# B&R Automation Studio project RobotNewEra (part 8)

### Data object Logical/MotionHandling/MotionInitFiles/SDC/sdc_j5_i (Ax)

#### sdc_j5_i.ax
```
InitParameter (Version=2.46.0, NcSwId=ACP10)
  ACP10AXIS_typ:
    dig_in:
      level:
        reference = ncACTIV_HI
        pos_hw_end = ncACTIV_HI
        neg_hw_end = ncACTIV_HI
        trigger1 = ncACTIV_HI
        trigger2 = ncACTIV_LO + ncQUICKSTOP
    encoder_if:
      parameter:
        count_dir = ncSTANDARD
        scaling:
          load:
            units = 360000
            rev_motor = 119
    limit:
      parameter:
        v_pos = 120000.0
        v_neg = 120000.0
        a1_pos = 240000.0
        a2_pos = 240000.0
        a1_neg = 240000.0
        a2_neg = 240000.0
        t_jolt = 0.1
        t_in_pos = 0.0
        pos_sw_end = 125000
        neg_sw_end = -125000
        ds_warning = 5000.0
        ds_stop = 10000.0
        a_stop = 1.0e+30
        dv_stop = 0.0
        dv_stop_mode = ncOFF
    controller:
      mode = ncPOSITION
      position:
        kv = 560.0
        tn = 0.0
        t_predict = 0.0004
        t_total = 0.0004
        p_max = 1.0e+30
        i_max = 20000.0
      speed:
        kv = 29.3
        tn = 0.0
        t_filter = 0.0
        isq_filter1:
          type = ncOFF
          a0 = 0.0
          a1 = 0.0
          b0 = 0.0
          b1 = 0.0
          b2 = 0.0
          c0_par_id = 0
          c1_par_id = 0
        isq_filter2:
          type = ncOFF
          a0 = 0.0
          a1 = 0.0
          b0 = 0.0
          b1 = 0.0
          b2 = 0.0
          c0_par_id = 0
          c1_par_id = 0
        isq_filter3:
          type = ncOFF
          a0 = 0.0
          a1 = 0.0
          b0 = 0.0
          b1 = 0.0
          b2 = 0.0
          c0_par_id = 0
          c1_par_id = 0
      uf:
        type = ncLINEAR
        auto_config = ncMOTOR_PAR
        u0 = 0.0
        un = 0.0
        fn = 50.0
        k_f_slip = 0.0
      ff:
        torque_load = 0.0
        torque_pos = 0.0
        torque_neg = 0.0
        kv_torque = 0.0
        inertia = 0.0
        t_filter_a = 0.0
    move:
      stop:
        parameter[0]:
          decel_ramp = ncA_LIMIT
          controller = ncON
        parameter[1]:
          decel_ramp = ncA_LIMIT
          controller = ncON
        parameter[2]:
          decel_ramp = ncA_LIMIT
          controller = ncON
        parameter[3]:
          decel_ramp = ncA_LIMIT
          controller = ncON
        quickstop:
          decel_ramp = ncA_LIMIT
        drive_error:
          decel_ramp = ncA_LIMIT
      homing:
        parameter:
          s = 0
          v_switch = 5000.0
          v_trigger = 500.0
          a = 50000.0
          mode = ncDIRECT
          edge_sw = ncPOSITIVE
          start_dir = ncPOSITIVE
          trigg_dir = ncPOSITIVE
          ref_pulse = ncOFF
          fix_dir = ncOFF
          tr_s_block = 0.0
          torque_lim = 0.0
          ds_block = 0.0
          ds_stop = 0.0
      basis:
        parameter:
          v_pos = 5000.0
          v_neg = 5000.0
          a1_pos = 100000.0
          a2_pos = 100000.0
          a1_neg = 100000.0
          a2_neg = 100000.0
    message:
      text:
        parameter:
          format = ncBREAK
          columns = 80
          data_modul = AcpError
```

### Data object Logical/MotionHandling/MotionInitFiles/SDC/sdc_j6_i (Ax)

#### sdc_j6_i.ax
```
InitParameter (Version=2.46.0, NcSwId=ACP10)
  ACP10AXIS_typ:
    dig_in:
      level:
        reference = ncACTIV_HI
        pos_hw_end = ncACTIV_HI
        neg_hw_end = ncACTIV_HI
        trigger1 = ncACTIV_HI
        trigger2 = ncACTIV_LO + ncQUICKSTOP
    encoder_if:
      parameter:
        count_dir = ncSTANDARD
        scaling:
          load:
            units = 360000
            rev_motor = 89
    limit:
      parameter:
        v_pos = 190000.0
        v_neg = 190000.0
        a1_pos = 380000.0
        a2_pos = 380000.0
        a1_neg = 380000.0
        a2_neg = 380000.0
        t_jolt = 0.1
        t_in_pos = 0.0
        pos_sw_end = 360000
        neg_sw_end = -360000
        ds_warning = 5000.0
        ds_stop = 10000.0
        a_stop = 1.0e+30
        dv_stop = 0.0
        dv_stop_mode = ncOFF
    controller:
      mode = ncPOSITION
      position:
        kv = 540.0
        tn = 0.0
        t_predict = 0.0004
        t_total = 0.0004
        p_max = 1.0e+30
        i_max = 2000.0
      speed:
        kv = 29.85
        tn = 0.0
        t_filter = 0.0
        isq_filter1:
          type = ncOFF
          a0 = 0.0
          a1 = 0.0
          b0 = 0.0
          b1 = 0.0
          b2 = 0.0
          c0_par_id = 0
          c1_par_id = 0
        isq_filter2:
          type = ncOFF
          a0 = 0.0
          a1 = 0.0
          b0 = 0.0
          b1 = 0.0
          b2 = 0.0
          c0_par_id = 0
          c1_par_id = 0
        isq_filter3:
          type = ncOFF
          a0 = 0.0
          a1 = 0.0
          b0 = 0.0
          b1 = 0.0
          b2 = 0.0
          c0_par_id = 0
          c1_par_id = 0
      uf:
        type = ncLINEAR
        auto_config = ncMOTOR_PAR
        u0 = 0.0
        un = 0.0
        fn = 50.0
        k_f_slip = 0.0
      ff:
        torque_load = 0.00094268
        torque_pos = 0.110223
        torque_neg = 0.100704
        kv_torque = 0.00253262
        inertia = 5.79039e-05
        t_filter_a = 0.0
    move:
      stop:
        parameter[0]:
          decel_ramp = ncA_LIMIT
          controller = ncON
        parameter[1]:
          decel_ramp = ncA_LIMIT
          controller = ncON
        parameter[2]:
          decel_ramp = ncA_LIMIT
          controller = ncON
        parameter[3]:
          decel_ramp = ncA_LIMIT
          controller = ncON
        quickstop:
          decel_ramp = ncA_LIMIT
        drive_error:
          decel_ramp = ncA_LIMIT
      homing:
        parameter:
          s = 0
          v_switch = 5000.0
          v_trigger = 500.0
          a = 50000.0
          mode = ncDIRECT
          edge_sw = ncPOSITIVE
          start_dir = ncPOSITIVE
          trigg_dir = ncPOSITIVE
          ref_pulse = ncOFF
          fix_dir = ncOFF
          tr_s_block = 0.0
          torque_lim = 0.0
          ds_block = 0.0
          ds_stop = 0.0
      basis:
        parameter:
          v_pos = 5000.0
          v_neg = 5000.0
          a1_pos = 100000.0
          a2_pos = 100000.0
          a1_neg = 100000.0
          a2_neg = 100000.0
    message:
      text:
        parameter:
          format = ncBREAK
          columns = 80
          data_modul = AcpError
```

### Data object Logical/MotionHandling/MotionInitFiles/robot_i (Cns) - ARNC0: CNC-System

- robot_i.cns (not shown)

### Package Logical/MotionHandling/Transformations - Trf Related

### Program Logical/MotionHandling/Transformations/Trf (ANSIC)

#### Trf.c - Implementation code
```c
/********************************************************************
 * COPYRIGHT -- Bernecker + Rainer
 ********************************************************************
 * Program: Trf
 * File: Trf.c
 * Author: frigenif
 * Created: December 08, 2011
 ********************************************************************
 * Implementation of program Trf
 ********************************************************************/

#include <bur/plctypes.h>
#include <TRF_LIB.h>

#ifdef _DEFAULT_INCLUDES
 #include <AsDefault.h>
#endif

void _INIT TrfINIT( void )
{

	/* Trasformation Configuration */

	/* Unit definintion */
	Robot_TRF.units.measure= TRF_DEGREES;
	Robot_TRF.units.epsilon= 0.000001;
	// Initialization
	// Warning: Delete those if = 0 then = ,they are only for Testpurpose
	if (HmiRetain.HmiRobot.CartesianLimits[0].Min == 0) HmiRetain.HmiRobot.CartesianLimits[0].Min = -2658;
	if (HmiRetain.HmiRobot.CartesianLimits[1].Min == 0) HmiRetain.HmiRobot.CartesianLimits[1].Min = -2658;
	if (HmiRetain.HmiRobot.CartesianLimits[2].Min == 0) HmiRetain.HmiRobot.CartesianLimits[2].Min = -602;
	if (HmiRetain.HmiRobot.CartesianLimits[0].Max == 0) HmiRetain.HmiRobot.CartesianLimits[0].Max = 2658;
	if (HmiRetain.HmiRobot.CartesianLimits[1].Max == 0) HmiRetain.HmiRobot.CartesianLimits[1].Max = 2658;
	if (HmiRetain.HmiRobot.CartesianLimits[2].Max == 0) HmiRetain.HmiRobot.CartesianLimits[2].Max = 3297;

	if (HmiRetain.HmiRobot.HomePos.Pos.x == 0) HmiRetain.HmiRobot.HomePos.Pos.x = 1854;
	if (HmiRetain.HmiRobot.HomePos.Pos.y == 0) HmiRetain.HmiRobot.HomePos.Pos.y = 0;
	if (HmiRetain.HmiRobot.HomePos.Pos.z == 0) HmiRetain.HmiRobot.HomePos.Pos.z = 1990;

	//	 Dimensions and position in the global coordinate system
	if (HmiRetain.HmiRobot.Mech[1].OffsetX == 0) HmiRetain.HmiRobot.Mech[1].OffsetX = 312.0;
	if (HmiRetain.HmiRobot.Mech[1].OffsetZ == 0) HmiRetain.HmiRobot.Mech[1].OffsetZ = 680.0;
	if (HmiRetain.HmiRobot.Mech[2].OffsetZ == 0) HmiRetain.HmiRobot.Mech[2].OffsetZ = 1075.0;
	if (HmiRetain.HmiRobot.Mech[3].OffsetX == 0) HmiRetain.HmiRobot.Mech[3].OffsetX = 400.0;
	if (HmiRetain.HmiRobot.Mech[3].OffsetZ == 0) HmiRetain.HmiRobot.Mech[3].OffsetZ = 235.0;
	if (HmiRetain.HmiRobot.Mech[4].OffsetX == 0) HmiRetain.HmiRobot.Mech[4].OffsetX = 882.0;
	if (HmiRetain.HmiRobot.Mech[5].OffsetX == 0) HmiRetain.HmiRobot.Mech[5].OffsetX = 260.0;

	Robot_TRF.mech.a0x = HmiRetain.HmiRobot.Mech[0].OffsetX;
	Robot_TRF.mech.a0y = HmiRetain.HmiRobot.Mech[0].OffsetY;
	Robot_TRF.mech.a0z = HmiRetain.HmiRobot.Mech[0].OffsetZ;
	Robot_TRF.mech.a1x = HmiRetain.HmiRobot.Mech[1].OffsetX;
	Robot_TRF.mech.a1y = HmiRetain.HmiRobot.Mech[1].OffsetY;
	Robot_TRF.mech.a1z = HmiRetain.HmiRobot.Mech[1].OffsetZ;
	Robot_TRF.mech.a2x = HmiRetain.HmiRobot.Mech[2].OffsetX;
	Robot_TRF.mech.a2y = HmiRetain.HmiRobot.Mech[2].OffsetY;
	Robot_TRF.mech.a2z = HmiRetain.HmiRobot.Mech[2].OffsetZ;
	Robot_TRF.mech.a3x = HmiRetain.HmiRobot.Mech[3].OffsetX;
	Robot_TRF.mech.a3y = HmiRetain.HmiRobot.Mech[3].OffsetY;
	Robot_TRF.mech.a3z = HmiRetain.HmiRobot.Mech[3].OffsetZ;
	Robot_TRF.mech.a4x = HmiRetain.HmiRobot.Mech[4].OffsetX;
	Robot_TRF.mech.a5x = HmiRetain.HmiRobot.Mech[5].OffsetX;

	Robot_TRF.mech.angles_type = TRF_CARDAN_ANGLES;

	/* preferred mode */
	Robot_TRF.mode.preferred = TRF_MODE_FRONT + TRF_MODE_CONVEX + TRF_MODE_POSITIVE;

	// Joint properties
	if (HmiRetain.HmiRobot.Mech[1].Direction == 0) HmiRetain.HmiRobot.Mech[1].Direction = 1;
	if (HmiRetain.HmiRobot.Mech[2].Direction == 0) HmiRetain.HmiRobot.Mech[2].Direction = 1;
	if (HmiRetain.HmiRobot.Mech[4].Direction == 0) HmiRetain.HmiRobot.Mech[4].Direction = 1;

	if (HmiRetain.HmiRobot.JointLimits[0].Min == 0) HmiRetain.HmiRobot.JointLimits[0].Min = -180;
	if (HmiRetain.HmiRobot.JointLimits[0].Max == 0) HmiRetain.HmiRobot.JointLimits[0].Max = 180;
	if (HmiRetain.HmiRobot.JointLimits[1].Min == 0) HmiRetain.HmiRobot.JointLimits[1].Min = -76;
	if (HmiRetain.HmiRobot.JointLimits[1].Max == 0) HmiRetain.HmiRobot.JointLimits[1].Max = 60;
	if (HmiRetain.HmiRobot.JointLimits[2].Min == 0) HmiRetain.HmiRobot.JointLimits[2].Min = -65; //-142;
	if (HmiRetain.HmiRobot.JointLimits[2].Max == 0) HmiRetain.HmiRobot.JointLimits[2].Max = 230;
	if (HmiRetain.HmiRobot.JointLimits[3].Min == 0) HmiRetain.HmiRobot.JointLimits[3].Min = -360;
	if (HmiRetain.HmiRobot.JointLimits[3].Max == 0) HmiRetain.HmiRobot.JointLimits[3].Max = 360; //-360;
	if (HmiRetain.HmiRobot.JointLimits[4].Min == 0) HmiRetain.HmiRobot.JointLimits[4].Min = -125;
	if (HmiRetain.HmiRobot.JointLimits[4].Max == 0) HmiRetain.HmiRobot.JointLimits[4].Max = 125;
	if (HmiRetain.HmiRobot.JointLimits[5].Min == 0) HmiRetain.HmiRobot.JointLimits[5].Min = -360;
	if (HmiRetain.HmiRobot.JointLimits[5].Max == 0) HmiRetain.HmiRobot.JointLimits[5].Max = 360;

	Robot_TRF.mech.axis_Q1.property = TRF_MATH_POSITIVE + HmiRetain.HmiRobot.Mech[0].Direction + TRF_SW_ENDS_ENABLE + TRF_MULT_FACTOR_DISABLE;
	Robot_TRF.mech.axis_Q1.min_sw_end = HmiRetain.HmiRobot.JointLimits[0].Min;
	Robot_TRF.mech.axis_Q1.max_sw_end = HmiRetain.HmiRobot.JointLimits[0].Max;
	Robot_TRF.mech.axis_Q1.maximal_change = 5000.0;	// obsolete
	Robot_TRF.mech.axis_Q1.mult_factor = 0.0;

	Robot_TRF.mech.axis_Q2.property = TRF_MATH_POSITIVE + HmiRetain.HmiRobot.Mech[1].Direction + TRF_SW_ENDS_ENABLE + TRF_MULT_FACTOR_DISABLE ;
	Robot_TRF.mech.axis_Q2.min_sw_end = HmiRetain.HmiRobot.JointLimits[1].Min;
	Robot_TRF.mech.axis_Q2.max_sw_end = HmiRetain.HmiRobot.JointLimits[1].Max;
	Robot_TRF.mech.axis_Q2.maximal_change = 5000.0;	// obsolete
	Robot_TRF.mech.axis_Q2.mult_factor = 0.0;

	Robot_TRF.mech.axis_Q3.property = TRF_MATH_POSITIVE + HmiRetain.HmiRobot.Mech[2].Direction + TRF_SW_ENDS_ENABLE + TRF_MULT_FACTOR_DISABLE;
	Robot_TRF.mech.axis_Q3.min_sw_end = HmiRetain.HmiRobot.JointLimits[2].Min;
	Robot_TRF.mech.axis_Q3.max_sw_end = HmiRetain.HmiRobot.JointLimits[2].Max;
	Robot_TRF.mech.axis_Q3.maximal_change = 5000.0;	// obsolete
	Robot_TRF.mech.axis_Q3.mult_factor = 0.0;

	Robot_TRF.mech.axis_Q4.property = TRF_MATH_POSITIVE + HmiRetain.HmiRobot.Mech[3].Direction + TRF_SW_ENDS_ENABLE + TRF_MULT_FACTOR_DISABLE;
	Robot_TRF.mech.axis_Q4.min_sw_end = HmiRetain.HmiRobot.JointLimits[3].Min;
	Robot_TRF.mech.axis_Q4.max_sw_end = HmiRetain.HmiRobot.JointLimits[3].Max;
	Robot_TRF.mech.axis_Q4.maximal_change = 5000.0;	// obsolete
	Robot_TRF.mech.axis_Q4.mult_factor = 0.0;

	Robot_TRF.mech.axis_Q5.property = TRF_MATH_POSITIVE + HmiRetain.HmiRobot.Mech[4].Direction + TRF_SW_ENDS_ENABLE + TRF_MULT_FACTOR_DISABLE;
	Robot_TRF.mech.axis_Q5.min_sw_end = HmiRetain.HmiRobot.JointLimits[4].Min;
	Robot_TRF.mech.axis_Q5.max_sw_end = HmiRetain.HmiRobot.JointLimits[4].Max;
	Robot_TRF.mech.axis_Q5.maximal_change = 5000.0;	// obsolete
	Robot_TRF.mech.axis_Q5.mult_factor = 0.0;

	Robot_TRF.mech.axis_Q6.property = TRF_MATH_POSITIVE + HmiRetain.HmiRobot.Mech[5].Direction + TRF_SW_ENDS_ENABLE + TRF_MULT_FACTOR_DISABLE;
	Robot_TRF.mech.axis_Q6.min_sw_end = HmiRetain.HmiRobot.JointLimits[5].Min;
	Robot_TRF.mech.axis_Q6.max_sw_end = HmiRetain.HmiRobot.JointLimits[5].Max;
	Robot_TRF.mech.axis_Q6.maximal_change = 5000.0;	// obsolete
	Robot_TRF.mech.axis_Q6.mult_factor = 0.0;

	/* Add link to dynamic model */
	RobotDynGeneric.addr_var_name = (UDINT)("OptMotion:Par6axATrf");
	Robot_TRF.ident.dyn_model = (UDINT)&(RobotDynGeneric);

	/* Pointers to transformation functions */
	Robot_TRF.fctaddr.direct = (UDINT) TRF_direct;
	Robot_TRF.fctaddr.inverse = (UDINT) TRF_inverse;
	Robot_TRF.fctaddr.get_mode = (UDINT) TRF_get_mode;

	/* Coupling between Axes*/
	if (HmiRetain.HmiRobot.Coupling[0].Enable == 0) HmiRetain.HmiRobot.Coupling[0].Enable = 1;
	if (HmiRetain.HmiRobot.Coupling[0].Coefficient == 0) HmiRetain.HmiRobot.Coupling[0].Coefficient = 1.0/120;
	if (HmiRetain.HmiRobot.Coupling[1].Enable == 0) HmiRetain.HmiRobot.Coupling[1].Enable = 1;
	if (HmiRetain.HmiRobot.Coupling[1].Coefficient == 0) HmiRetain.HmiRobot.Coupling[1].Coefficient = -1.0/89;

	ExtJoint.link[0].enabled = HmiRetain.HmiRobot.Coupling[0].Enable;
	ExtJoint.link[0].idealToCpl = 0;
	ExtJoint.link[0].i = 4;
	ExtJoint.link[0].j = 3; // 4 Affects 5
	ExtJoint.link[0].coeff = HmiRetain.HmiRobot.Coupling[0].Coefficient;

	ExtJoint.link[1].enabled = HmiRetain.HmiRobot.Coupling[1].Enable;
	ExtJoint.link[1].idealToCpl = 0;
	ExtJoint.link[1].i = 5;
	ExtJoint.link[1].j = 4; // 5 Affects 6
	ExtJoint.link[1].coeff = HmiRetain.HmiRobot.Coupling[1].Coefficient;

	ExtJoint.link[2].enabled = HmiRetain.HmiRobot.Coupling[2].Enable;
	ExtJoint.link[2].idealToCpl = 0;
	ExtJoint.link[2].i = 5;
	ExtJoint.link[2].j = 3; // 4 Affects 6
	ExtJoint.link[2].coeff = HmiRetain.HmiRobot.Coupling[2].Coefficient;

	ExtTrfData.joint = &ExtJoint;
	Robot_TRF.type_04 = &ExtTrfData;

	/* Initialization of transformation object */
	TRF_6AX_InitStatus = TRF_init_instance((UDINT)"Robot_TRF");

}

void _CYCLIC TrfCYCLIC( void )
{

	if (AxesAddress != 0)
	{
		pAxes = (Axes_Type*) AxesAddress;

		/* call direct tranformations to allign TCP axes when homing */
		TrfInPos[0]	=	(LREAL) (*pAxes)[AXIS_Q1].Output.Monitor.Position;
		TrfInPos[1]	=	(LREAL) (*pAxes)[AXIS_Q2].Output.Monitor.Position;
		TrfInPos[2]	=	(LREAL) (*pAxes)[AXIS_Q3].Output.Monitor.Position;
		TrfInPos[3]	=	(LREAL) (*pAxes)[AXIS_Q4].Output.Monitor.Position;
		TrfInPos[4]	=	(LREAL) (*pAxes)[AXIS_Q5].Output.Monitor.Position;
		TrfInPos[5]	=	(LREAL) (*pAxes)[AXIS_Q6].Output.Monitor.Position;

		SimPos[0]	=	(*pAxes)[AXIS_Q1].Output.Monitor.Position;
		SimPos[1]	=	(*pAxes)[AXIS_Q2].Output.Monitor.Position;
		SimPos[2]	=	(*pAxes)[AXIS_Q3].Output.Monitor.Position;
		SimPos[3]	=	(*pAxes)[AXIS_Q4].Output.Monitor.Position;
		SimPos[4]	=	(*pAxes)[AXIS_Q5].Output.Monitor.Position;
		SimPos[5]	=	(*pAxes)[AXIS_Q6].Output.Monitor.Position;

		TrfInPosExt[0]	= 0;
		TrfInPosExt[1]	= 0;
		TrfInPosExt[2]	= 0;
		TrfInPosExt[3]	= 0;
		TrfInPosExt[4]	= 0;
		TrfInPosExt[5]	= 0;

		TrfDirectTransStatus = TRF_direct(&Robot_TRF, (UDINT)&TrfInPos[0], (UDINT)&TrfInPosExt[0], (UDINT)&TrfOutPos[0],(UDINT) &TrfDirectInfo[0]);

		(*pAxes)[AXIS_X].Input.Parameter.AutoPosition	= (REAL) (TrfOutPos[0]);
		(*pAxes)[AXIS_Y].Input.Parameter.AutoPosition	= (REAL) (TrfOutPos[1]);
		(*pAxes)[AXIS_Z].Input.Parameter.AutoPosition	= (REAL) (TrfOutPos[2]);
		(*pAxes)[AXIS_A].Input.Parameter.AutoPosition	= (REAL) (TrfOutPos[3]);
		(*pAxes)[AXIS_B].Input.Parameter.AutoPosition	= (REAL) (TrfOutPos[4]);
		(*pAxes)[AXIS_C].Input.Parameter.AutoPosition	= (REAL) (TrfOutPos[5]);

		(*pAxes)[AXIS_X].Input.Parameter.HomePosition	= (REAL) (TrfOutPos[0]);
		(*pAxes)[AXIS_Y].Input.Parameter.HomePosition	= (REAL) (TrfOutPos[1]);
		(*pAxes)[AXIS_Z].Input.Parameter.HomePosition	= (REAL) (TrfOutPos[2]);
		(*pAxes)[AXIS_A].Input.Parameter.HomePosition	= (REAL) (TrfOutPos[3]);
		(*pAxes)[AXIS_B].Input.Parameter.HomePosition	= (REAL) (TrfOutPos[4]);
		(*pAxes)[AXIS_C].Input.Parameter.HomePosition	= (REAL) (TrfOutPos[5]);

		(*pAxes)[AXIS_Q1].Output.Monitor.DecoupledPosition = (*pAxes)[AXIS_Q1].Output.Monitor.Position;
		(*pAxes)[AXIS_Q2].Output.Monitor.DecoupledPosition = (*pAxes)[AXIS_Q2].Output.Monitor.Position;
		(*pAxes)[AXIS_Q3].Output.Monitor.DecoupledPosition = (*pAxes)[AXIS_Q3].Output.Monitor.Position;
		(*pAxes)[AXIS_Q4].Output.Monitor.DecoupledPosition = (*pAxes)[AXIS_Q4].Output.Monitor.Position;
		(*pAxes)[AXIS_Q5].Output.Monitor.DecoupledPosition = (*pAxes)[AXIS_Q5].Output.Monitor.Position - (*pAxes)[AXIS_Q4].Output.Monitor.Position * HmiRetain.HmiRobot.Coupling[0].Coefficient * ((LREAL) HmiRetain.HmiRobot.Coupling[0].Enable) ;
		(*pAxes)[AXIS_Q6].Output.Monitor.DecoupledPosition = (*pAxes)[AXIS_Q6].Output.Monitor.Position - (*pAxes)[AXIS_Q5].Output.Monitor.Position * HmiRetain.HmiRobot.Coupling[1].Coefficient * ((LREAL) HmiRetain.HmiRobot.Coupling[1].Enable)
			- (*pAxes)[AXIS_Q4].Output.Monitor.Position * HmiRetain.HmiRobot.Coupling[2].Coefficient * ((LREAL) HmiRetain.HmiRobot.Coupling[2].Enable);

		SimPosVisu[0]	=	(*pAxes)[AXIS_Q1].Output.Monitor.DecoupledPosition;
		SimPosVisu[1]	=	(*pAxes)[AXIS_Q2].Output.Monitor.DecoupledPosition;
		SimPosVisu[2]	=	(*pAxes)[AXIS_Q3].Output.Monitor.DecoupledPosition;
		SimPosVisu[3]	=	(*pAxes)[AXIS_Q4].Output.Monitor.DecoupledPosition;
		SimPosVisu[4]	=	(*pAxes)[AXIS_Q5].Output.Monitor.DecoupledPosition;
		SimPosVisu[5]	=	(*pAxes)[AXIS_Q6].Output.Monitor.DecoupledPosition;
	}

}
```

#### TrfPrv.var - Local variables
```iecst
(********************************************************************
 * COPYRIGHT -- Bernecker + Rainer
 ********************************************************************
 * Program: Trf
 * File: Trf.var
 * Author: frigenif
 * Created: December 08, 2011
 ********************************************************************
 * Local variables of program Trf
 ********************************************************************)
VAR
	TRF_6AX_InitStatus : UDINT;
	pAxes : REFERENCE TO ARRAY[0..MAX_AX_MINUS_ONE] OF Axes_Type;
	AxesAddress : UDINT := 0;
	TrfOutPos : ARRAY[0..5] OF LREAL;
	TrfInPos : ARRAY[0..5] OF LREAL;
	TrfInPosExt : ARRAY[0..5] OF LREAL;
	TrfDirectInfo : ARRAY[0..1] OF UDINT;
	TrfDirectTransStatus : UDINT;
	SimPosVisu : ARRAY[0..5] OF REAL;
	SimPos : ARRAY[0..5] OF REAL;
	RobotDynGeneric : TRF_DYN_typ := (0);
	ExtJoint : TRF_extEntity_t := (0);
	ExtTrfData : TRF_EXT_typ := (0);
END_VAR
```

### Package Logical/MotionHandling/Interpreter - Interpreter xml config files

### Data object Logical/MotionHandling/Interpreter/GmcIpConfig/gmcipsys (Cnc, version 2.47.4)

#### gmcipsys.cnc
```
LANGS (defaultLangId=3, defaultDataLangId=3)
  CMDQUEUE (BufferSize=15)
  MEM (ReserveMB=5, LimitPercent=80%)
  EXEC (InstrBurstBG=200, CycleBurstBG=0, Stack=16384, MinorStack=2048, EStack=1024)
  LOAD (ReadLineBurstMax=100, ReadLineBurstMin=20, ParseLineBurstMax=10, ParseLineBurstMin=2, RuntimeIOBlocking=No)
  DISABLE_MSG = 15238 
    15336 
    15337 
    15666 
    15784 
    15864 
    15740
  LANG (langId=1, langName=B&R GCode, langModule=ailgcode)
    LANGCONFIG gmciplbr
    LANGCONFIG gmcipcbr
    LANGCONFIG gmcipubr
    FILEEXT .cnc
    FILEEXT .prg
    MAINSEARCHPATH $ (FileDevice=CNC_PrgDir)
    MAINSEARCHPATH $ (DataObject=Yes)
    INCLUDEPATH $ (FileDevice=CNC_PrgDir)
    INCLUDEPATH $ (DataObject=Yes)
  LANG (langId=2, langName=Alternative Language 1 GCode, langModule=ailgcode)
    LANGCONFIG gmciplsm
    LANGCONFIG gmcipcbr
    LANGCONFIG gmcipcsm
    LANGCONFIG gmcipusm
    FILEPREFIX = _N_
    FILEEXT = .MPF
    FILEEXT = _MPF
    FILEEXT = .SPF
    FILEEXT = _SPF
    MAINSEARCHPATH = \$ (FileDevice=CNC_PrgDir)
    MAINSEARCHPATH = \_N_MPF_DIR\$ (FileDevice=CNC_PrgDir)
    MAINSEARCHPATH = \_N_SPF_DIR\$ (FileDevice=CNC_PrgDir)
    MAINSEARCHPATH = $ (DataObject=1)
    INCLUDEPATH = \$ (FileDevice=CNC_PrgDir)
    INCLUDEPATH = \_N_SPF_DIR\$ (FileDevice=CNC_PrgDir)
    INCLUDEPATH = \_N_MPF_DIR\$ (FileDevice=CNC_PrgDir)
    INCLUDEPATH = $ (DataObject=1)
  LANG (langId=3, langName=IEC-ST, langModule=ailgcode)
    LANGCONFIG gmcipiec
    LANGCONFIG gmcipmx (RequireFnIgnore=MXConvertOrient)
    FILEEXT .typ (DeclScope=IP_GLOBAL)
    FILEEXT .var (DeclScope=IP_GLOBAL)
    FILEEXT .fun (DeclScope=IP_GLOBAL)
    FILEEXT .iec (DeclScope=IP_LOCAL)
    FILEEXT .st (DeclScope=IP_LOCAL)
    FILEEXT _iec (DeclScope=IP_LOCAL)
    MAINSEARCHPATH = \$ (FileDevice=IEC_PrgDir)
    MAINSEARCHPATH = \$ (FileDevice=CNC_PrgDir)
    MAINSEARCHPATH \TYP\$ (FileDevice=CNC_PrgDir, DataObject=No)
    MAINSEARCHPATH = $ (DataObject=1)
    INCLUDEPATH = \$ (FileDevice=IEC_PrgDir)
    INCLUDEPATH = \$ (FileDevice=CNC_PrgDir)
    INCLUDEPATH \TYP\$ (FileDevice=CNC_PrgDir, DataObject=No)
    INCLUDEPATH = $ (DataObject=1)
  XML_INCLUDE gmcipus (IfNotExist=Warn)
```

### Data object Logical/MotionHandling/Interpreter/GmcIpConfig/gmciplbr (Cnc, version 2.47.4)

#### gmciplbr.cnc
```
Root (LangModule=ailgcode, Version=1.0)
  BuiltInProcs:
    cancel = beginpathsynch
        StopCyclicGroups(:${*}:);
      endpathsynch (MinArgs=1, MaxArgs=*)
  BuiltInFns (PatternSuffix=:\[)
    ABS = Abs(:$[1]:) (NumArgs=1, Inline=Yes)
    SQR = ($[1] * $[1]) (NumArgs=1)
    ACOS = ACos(:$[1]:) (NumArgs=1, Inline=Yes)
    ASIN = ASin(:$[1]:) (NumArgs=1, Inline=Yes)
    ATAN = ATan(:$[1]:) (NumArgs=1, Inline=Yes)
    COS = Cos(:$[1]:) (NumArgs=1, Inline=Yes)
    DEXP = DExp(:$[1]:) (NumArgs=1, Inline=Yes)
    EXP = Exp(:$[1]:) (NumArgs=1, Inline=Yes)
    FIX = Fix(:$[1]:) (NumArgs=1, Inline=Yes)
    FRACT = Fract(:$[1]:) (NumArgs=1, Inline=Yes)
    FUP = Fup(:$[1]:) (NumArgs=1, Inline=Yes)
    INV = ~($[1]) (NumArgs=1, Inline=Yes)
    LN = Ln(:$[1]:) (NumArgs=1, Inline=Yes)
    LOG = Log(:$[1]:) (NumArgs=1, Inline=Yes)
    ROUND = ToInt(:$[1]:) (NumArgs=1, Inline=Yes)
    SIN = Sin(:$[1]:) (NumArgs=1, Inline=Yes)
    SQRT = Sqrt(:$[1]:) (NumArgs=1, Inline=Yes)
    TAN = Tan(:$[1]:) (NumArgs=1, Inline=Yes)
    BOOL = ToBool(:$[1]:) (NumArgs=1, Inline=Yes)
    INT = Fix(:$[1]:) (NumArgs=1, Inline=Yes)
    ADR = Adr(:\$[1]:) (NumArgs=1, Inline=Yes)
    SIZEOF = Sizeof(:\$[1]:) (NumArgs=1, Inline=Yes)
    NUM_LOADED_FILES = NumLoadedFiles(::) (NumArgs=0)
    NUM_LOADED_PROG_FILES = NumLoadedProgFiles(::) (NumArgs=0)
    MEM_SIZE_IP_ALL = MemSizeIpInstAll(::) (NumArgs=0)
    MEM_SIZE_IP_LIB = MemSizeIpInst(::) (NumArgs=0)
    MEM_SIZE_SHLIB = MemSizeShLib(::) (NumArgs=0)
    MEM_SIZE_FILE = MemSizeFile(:$[1]:) (MinArgs=0, MaxArgs=1)
    MEM_SIZE_IP_STACK_SPACE = MemStackSpace(::) (NumArgs=0)
  AxesSpec:
    AxisRef = $\s*=\s*AC (Mode=3)
    AxisRef = $\s*=\s*IC (Mode=4)
  PVMacros:
    RDISABLE (ArrayDims=0, Group=500)
      CALL = @#job->sa.keep_alive = 1;
        @#thread.sa_keep_alive = 1; (Inline=Yes)
  Parameters:
    R (IndexType=RParamIndex, ValueType=FLOAT)
      ARG (ref=EXPR, DataType=RParamIndex)
    P (IndexType=RParamIndex, ValueType=FLOAT)
      ARG (ref=EXPR, DataType=RParamIndex)
    EXB (IndexType=EXParamIndex, ValueType=Byte)
      ARG (ref=EXPR, DataType=EXParamIndex)
    EXW (IndexType=EXParamIndex, ValueType=Word)
      ARG (ref=EXPR, DataType=EXParamIndex)
    EXL (IndexType=EXParamIndex, ValueType=Long)
      ARG (ref=EXPR, DataType=EXParamIndex)
    EXF (IndexType=EXFParamIndex, ValueType=FLOAT)
      ARG (ref=EXPR, DataType=EXFParamIndex)
    MW (Synchronous=Yes, IndexType=MParamIndex, ValueType=Word)
      ARG (ref=EXPR, DataType=MParamIndex)
    ML (Synchronous=Yes, IndexType=MParamIndex, ValueType=Long)
      ARG (ref=EXPR, DataType=MParamIndex)
    MF (Synchronous=Yes, IndexType=MParamIndex, ValueType=FLOAT)
      ARG (ref=EXPR, DataType=MParamIndex)
  PrimTypes (PatternSuffix=:[^\[], MapIECTypes=Yes)
  Preprocess:
    PP_RULE_FRAME_I (Search=$FRAME_I, Replace=[1,0,0,0,1,0,0,0,1,0,0,0])
    PP_RULE_FRAME_DEF (Search=FRAME, Replace=LREAL{12})
  FubTemplates:
    StdFubTemplate (IsDefault=Yes, Inline=Yes)
      Arg (ref=FUBINST, DataType=FLOAT)
      Arg (ref=FUBERRLEV, DataType=FLOAT)
      Arg (ref=PATHSYNCH, DataType=FLOAT)
      Arg (ref=BLOCKING, DataType=FLOAT)
  SynchActions:
    SABlocks:
      default (IsDefault=Yes)
        cyclic (Inline=Yes)
          Arg (ref=ACTIONS, DataType=STATEMENTS)
          Arg (ref=ID, DataType=FLOAT, DefaultInt=-1, MinCount=0, MaxCount=1)
      whenever:
        cyclic (Inline=Yes)
          Arg (ref=COND, DataType=FLOAT)
          Arg (ref=ACTIONS, DataType=STATEMENTS)
          Arg (ref=ID, DataType=FLOAT, DefaultInt=-1, MinCount=0, MaxCount=1)
      when:
        cyclic (Inline=Yes)
          Arg (ref=COND, DataType=FLOAT)
          Arg (ref=ACTIONS, DataType=STATEMENTS)
          Arg (ref=ID, DataType=FLOAT, DefaultInt=-1, MinCount=0, MaxCount=1)
      every:
        cyclic (Inline=Yes)
          Arg (ref=COND, DataType=FLOAT)
          Arg (ref=ACTIONS, DataType=STATEMENTS)
          Arg (ref=ID, DataType=FLOAT, DefaultInt=-1, MinCount=0, MaxCount=1)
      from:
        cyclic (Inline=Yes)
          Arg (ref=COND, DataType=FLOAT)
          Arg (ref=ACTIONS, DataType=STATEMENTS)
          Arg (ref=ID, DataType=FLOAT, DefaultInt=-1, MinCount=0, MaxCount=1)
    NonModalActivation:
      Start = @#thread.sa_last_keep_alive = 1;
        ActivateCyclicGroup(:-1:);
      Stop = WaitStopCyclicGroups(:(:-1:):);
  ParserData (NestedComments=Yes, DefaultCaseSensitive=No, CommentsSpanLines=No, SubDeclsLocalToFile=Yes, ProgDeclsLocalToFile=Yes, AllowUnprefixedFileCalls=No, LocalVarScopeForMainProg=No, FileScopeVarsVisibleInSub=Yes, MainPrgReturnAtNextMainPrgHdr=Yes, MaxSizePassByValue=1024, AllowVarReadBeforeAssign=No, AllowArrayRefWithoutIndex=Yes, AllowStructMemberAutoDereference=Yes, AllowVariableAutoDereference=Yes, AllowIgnoredExtraSubArgs=Yes, EnableStringCharacterIndexing=Yes, OnMacroRedefinition=Warn, CheckFileTimestampBeforeCalls=Yes)
    TKG_END_OF_LINE = \n (IsPattern=No)
    TKG_LINE_CONTINUE = \ (IsPattern=No, FileXLInvalid=Yes)
    TKG_LINE_BREAK = @@
    TKG_ARITH_BINARY_MODULO = MOD
    TKG_TRUE = TRUE:\W (IsPattern=Yes)
    TKG_FALSE = FALSE:\W (IsPattern=Yes)
    TKG_PAREVAL_MODAL_ID = ID:[\s=] (FileXLInvalid=Yes, IsPattern=Yes)
    TKG_OPEN_COMMENT = (
    TKG_CLOSE_COMMENT = )
    TKG_OPEN_BRACKET = [
    TKG_COMMA = ,
    TKG_CLOSE_BRACKET = ]
    TKG_OPEN_INDEXBRACKET = {
    TKG_CLOSE_INDEXBRACKET = }
    TKG_NUMBER = \d+\.\d+|\d+\.:[^\.] (IsPattern=Yes)
    TKG_INTEGER = \d+ (IsPattern=Yes)
    TKG_FRACTION = \.\d+ (IsPattern=Yes)
    TKG_DOT = \.:\w (IsPattern=Yes, FollowedBy=TKG_STRUCT_MEMBER_REF)
    TKG_STRUCT_MEMBER_REF = \w|\w[\w\d]+ (IsPattern=Yes, Restricted=Yes)
    TKG_NUMBER_EXP = EX:[\s\d\+\-\.] (IsPattern=Yes)
    TKG_MACRO_DEFINE_GLOBAL = define\s+ip_global:\s (IsPattern=Yes, FollowedBy=TKG_MACRO_NAME)
    TKG_MACRO_DEFINE = define\s+local:\s|define:\s (IsPattern=Yes, FollowedBy=TKG_MACRO_NAME)
    TKG_MACRO_UNDEFINE = undefine:\s (IsPattern=Yes, FollowedBy=TKG_MACRO_NAME)
    TKG_MACRO_AS = as:[\s\n] (IsPattern=Yes, FollowedBy=TKG_MACRO_TEXT)
    TKG_MACRO_NAME = [$\w][$\w\d]+ (Restricted=Yes, IsPattern=Yes)
    TKG_MACRO_TEXT = . (Restricted=Yes, IsPattern=Yes)
    TKG_BUILTIN_NUM_FN_NAME
    _TKG_LABEL_DEF1:
      TKG_LABEL_DEF = L[\w\d]+:\:[^\w\d] (IsPattern=Yes, FollowedBy=TKG_LABEL_SUFFIX)
    TKG_SUBPROG_START = %:L (FileXLInvalid=Yes, IsPattern=Yes, FollowedBy=TKG_SUBPROG_NAME)
    TKG_SUBPROG_NAME = L\d+ (IsPattern=Yes, Restricted=Yes)
    TKG_SUBPROG_CALL = L:L\d (IsPattern=Yes, FollowedBy=TKG_SUBPROG_NAME)
    TKG_SUBPROG_PROTO = %D:L (IsPattern=Yes, FollowedBy=TKG_SUBPROG_NAME)
    TKG_SUBCALL_REPEAT_PREFIX = O:[\s\d] (IsPattern=Yes, FollowedBy=TKG_INTEGER)
    TKG_EXTERN = EXTERN:\s (IsPattern=Yes, FollowedBy=TKG_PROG_FILE_NAME)
    TKG_ARG_PASSBYREF = VAR\s (IsPattern=Yes)
    TKG_SET_MODAL_SUB = MCALL:\W (FileXLInvalid=Yes, IsPattern=Yes)
    TKG_PROG_START = %:\d (IsPattern=Yes, FollowedBy=TKG_PROG_NAME)
    TKG_PROG_NAME = \d+ (IsPattern=Yes, Restricted=Yes)
    TKG_PROG_CALL = L:[^L] (IsPattern=Yes, FollowedBy=TKG_PROG_FILE_NAME)
    TKG_PROG_FILE_NAME = [\^#&@']?[\w\d\.\\]+:[^\w\d\.\\\:]|[\^#][\w\d]+\:[\w\d\.\\]+ (IsPattern=Yes, Restricted=Yes)
    TKG_SUPPRESS_SINGLE_STEP = NOHALT
    TKG_NC_BLOCK_PREFIX = N:[\d\s] (IsPattern=Yes)
    TKG_PARAM_PREFIX = R:\d|P:\d|M[WLF]:\d|EX[WLBF]:\d (IsPattern=Yes)
    TKG_SUBRANGE = ..
    TKG_G_CODE_PREFIX = G:[\s\d] (IsPattern=Yes)
    TKG_M_CODE_PREFIX = M:[\s\d\[] (IsPattern=Yes)
    TKG_PAREVAL_DO = do:\s (FileXLInvalid=Yes, IsPattern=Yes)
    TKG_GOTO = $GOTO:\s (FileXLInvalid=Yes, IsPattern=Yes, OptFollowedBy=TKG_GOTO_DEST)
    TKG_GOTO_DEST = \w[\w\d]* (IsPattern=Yes, Restricted=Yes)
    TKG_LOGICAL_BINARY_AND = &&
    TKG_LOGICAL_BINARY_OR = ||
    TKG_LOGICAL_BINARY_XOR = XOR
    TKG_STRING_CONCAT = <<
    TKG_COMP_BINARY_GREATER_THAN_OR_EQ = >=
    TKG_COMP_BINARY_LESS_THAN_OR_EQ = <=
    TKG_COMP_BINARY_EQUAL_TO = ==
    TKG_COMP_BINARY_NOT_EQUAL_TO = !=
    TKG_COMP_BINARY_GREATER_THAN = >
    TKG_COMP_BINARY_LESS_THAN = <
    TKG_ASSIGN_EQ = =
    TKG_LOGICAL_UNARY_NOT = !
    TKG_BITWISE_BINARY_AND = &
    TKG_BITWISE_BINARY_OR = |
    TKG_BITWISE_BINARY_XOR = ^
    TKG_BITWISE_UNARY_COMPLEMENT = ~
    TKG_ARITH_BINARY_PLUS = +
    TKG_ARITH_BINARY_MINUS = -
    TKG_ARITH_BINARY_POWER = **
    TKG_ARITH_BINARY_MULTIPLY = *
    TKG_ARITH_BINARY_DIVIDE = /
    TKG_IF = $IF (FileXLInvalid=Yes)
    TKG_THEN = $THEN (FileXLInvalid=Yes)
    TKG_BLOCK_ELSEIF = $ELSEIF (FileXLInvalid=Yes)
    TKG_BLOCK_ELSE = $ELSE (FileXLInvalid=Yes)
    TKG_BLOCK_ENDIF = $ENDIF (FileXLInvalid=Yes)
    TKG_SWITCH = $SWITCH (FileXLInvalid=Yes)
    TKG_SWITCH_CASE = $CASE (FileXLInvalid=Yes)
    TKG_SWITCH_DEFAULT = $DEFAULT (FileXLInvalid=Yes)
    TKG_ENDSWITCH = $ENDSWITCH (FileXLInvalid=Yes)
    TKG_FOR = $FOR (FileXLInvalid=Yes)
    TKG_ENDFOR = $ENDFOR (FileXLInvalid=Yes)
    TKG_WHILE = $WHILE (FileXLInvalid=Yes)
    TKG_ENDWHILE = $ENDWHILE (FileXLInvalid=Yes)
    TKG_DO = $DO (FileXLInvalid=Yes)
    TKG_ENDDO = $ENDDO (FileXLInvalid=Yes)
    TKG_BREAK = $BREAK (FileXLInvalid=Yes)
    TKG_CONTINUE = $CONTINUE (FileXLInvalid=Yes)
    TKG_PRIM_TYPE (IsPattern=Yes)
    TKG_PV_DECL = def:\s (IsPattern=Yes)
    TKG_PV_UNDECL = ~def:\s (IsPattern=Yes)
    TKG_PV_DECL_REF = \w[\w\d\.\:\*]+|\w (IsPattern=Yes, Restricted=Yes)
    TKG_VARSCOPE_IP_LOCAL = local:[\s\n] (IsPattern=Yes)
    TKG_VARSCOPE_IP_GLOBAL = ip_global:[\s\n] (IsPattern=Yes)
    TKG_VARSCOPE_NC_GLOBAL = nc_global:[\s\n] (IsPattern=Yes)
    TKG_VARSCOPE_PLC_GLOBAL = plc_global:[\s\n] (IsPattern=Yes)
    TKG_VAR_RETAIN = retain:\s (IsPattern=Yes)
    TKG_VARSYNCH_IP = ip_synch:\s (IsPattern=Yes)
    TKG_VARSYNCH_PATH = path_synch:\s (IsPattern=Yes)
    TKG_LABEL_DEF = \w:\:|\w[\w\d]+:\: (IsPattern=Yes, FollowedBy=TKG_LABEL_SUFFIX)
    TKG_LABEL_SUFFIX = : (Restricted=Yes)
    TKG_FUB_DECL = fub:\s (IsPattern=Yes)
    TKG_FUB_ERR_LEV_1 = error_level_1:\s (IsPattern=Yes)
    TKG_FUB_ERR_LEV_2 = error_level_2:\s (IsPattern=Yes)
    TKG_FUB_ERR_LEV_3 = error_level_3:\s (IsPattern=Yes)
    TKG_FUB_ERR_LEV_4 = error_level_4:\s (IsPattern=Yes)
    TKG_FUB_BLOCKING = blocking:\s (IsPattern=Yes)
    TKG_FUB_NON_BLOCKING = non_blocking:\s (IsPattern=Yes)
    TKG_IEC_TYPED_VALUE = #[\w\d]+ (IsPattern=Yes)
    TKG_REFERENCE = ref:[\s\n]|reference:[\s\n] (IsPattern=Yes, FollowedBy=TKG_IEC_TO)
    TKG_IEC_TO = to:[\s\n] (IsPattern=Yes, Restricted=Yes)
    TKG_ACCESS = ACCESS:[\s\n] (IsPattern=Yes)
    TKG_WORD = \w|\w[\w\d\.]+ (IsPattern=Yes)
  StringChars (AsciiStringStart=", UTF16StringStart=W", UTF16StringEnd=")
    EscapeSeq (Search=$N, ReplaceValue=10)
    EscapeSeq (Search=$L, ReplaceValue=10)
    EscapeSeq (Search=$P, ReplaceValue=12)
    EscapeSeq (Search=$R, ReplaceValue=13)
    EscapeSeq (Search=$T, ReplaceValue=9)
    EscapeSeq (Search=$Q, ReplaceStr=")
    EscapeSeq (Search=$', ReplaceStr=')
    EscapeSeq (Search=$", ReplaceStr=")
    EscapeSeq (Search=$[\dA-Fa-f]+, IsPattern=Yes, ReplaceEncodingBase=16)
    EscapeSeq (Search=$$, ReplaceStr=$)
    EscapeSeq (Search=$, ReplaceStr=)
```

### Data object Logical/MotionHandling/Interpreter/GmcIpConfig/gmcipcbr (Cnc, version 2.47.4)

- gmcipcbr.cnc (not shown)

### Data object Logical/MotionHandling/Interpreter/GmcIpConfig/gmciplsm (Cnc, version 2.47.4)

#### gmciplsm.cnc
```
Root (LangModule=ailgcode, Version=1.0)
  PrimTypes (CaseSensitive=No)
    REAL (BRType=LREAL)
    INT (BRType=DINT)
    CHAR (BRType=USINT)
    BOOL (BRType=BOOL)
    STRING (BRType=STRING)
    AXIS (BRType=AXIS)
    BR_LREAL (BRType=LREAL)
    BR_REAL (BRType=REAL)
    BR_UDINT (BRType=UDINT)
    BR_DINT (BRType=DINT)
    BR_UINT (BRType=UINT)
    BR_INT (BRType=INT)
    BR_USINT (BRType=USINT)
    BR_SINT (BRType=SINT)
    BR_BOOL (BRType=BOOL)
    BR_TIME (BRType=TIME)
    BR_DATE_AND_TIME (BRType=DATE_AND_TIME)
  Preprocess:
    PP_RULE_NCK (Search=NCK , Replace=nc_global )
    PP_RULE_CHAN (Search=CHAN , Replace=ip_global )
    PP_RULE_FRAME_I (Search=$FRAME_I, Replace=(1,0,0,0,1,0,0,0,1,0,0,0))
    PP_RULE_FRAME_DEF (Search=FRAME, Replace=REAL[12])
  BuiltInProcs:
    cancel = beginpathsynch
        StopCyclicGroups(:${*}:);
      endpathsynch (MinArgs=1, MaxArgs=*)
    RET = #next_motion.Command = MPCMD_SET_M_FCT;
      #next_motion.Data.I4_value = 17;
      PushPacket(::);
      ReturnTo(:${*}:); (MinArgs=0, MaxArgs=4, Eval=Early, Inline=Yes)
  BuiltInFns:
    ABS = Abs(:$[1]:) (NumArgs=1, Inline=Yes)
    SIN = Sin(:$[1]:) (NumArgs=1, Inline=Yes)
    COS = Cos(:$[1]:) (NumArgs=1, Inline=Yes)
    TAN = Tan(:$[1]:) (NumArgs=1, Inline=Yes)
    ASIN = ASin(:$[1]:) (NumArgs=1, Inline=Yes)
    ACOS = ACos(:$[1]:) (NumArgs=1, Inline=Yes)
    ATAN = ATan(:$[1]:) (NumArgs=1, Inline=Yes)
    ATAN2 = ATan2(:$[1],$[2]:) (NumArgs=2, Inline=Yes)
    SQRT = Sqrt(:$[1]:) (NumArgs=1, Inline=Yes)
    POT = (($[1])*($[1])) (NumArgs=1, Inline=Yes)
    TRUNC = Fix(:$[1]:) (NumArgs=1, Inline=Yes)
    ROUND = Round(:$[1]:) (NumArgs=1, Inline=Yes)
    LN = Ln(:$[1]:) (NumArgs=1, Inline=Yes)
    EXP = Exp(:$[1]:) (NumArgs=1, Inline=Yes)
    MINVAL = MinVal(:$[1], $[2]:) (NumArgs=2, Inline=Yes)
    MAXVAL = MaxVal(:$[1], $[2]:) (NumArgs=2, Inline=Yes)
    BOUND = Bounds(:$[1], $[2], $[3]:) (NumArgs=3, Inline=Yes)
    TO_BOOL = ToBool(:$[1]:) (NumArgs=1, Inline=Yes)
    TO_INT = ToInt(:$[1]:) (NumArgs=1, Inline=Yes)
    TO_CHAR = ToChar(:$[1]:) (NumArgs=1, Inline=Yes)
    TO_REAL = ToLReal(:$[1]:) (NumArgs=1, Inline=Yes)
    TO_FLOAT = ToFloat(:$[1]:) (NumArgs=1, Inline=Yes)
    DEFINED = Defined(:$[1]:) (NumArgs=1, Inline=Yes)
    TIME_MS = TimeMs(::) (NumArgs=0)
    SET = ${*} (MinArgs=0, MaxArgs=*, Inline=Yes)
    REP = ArrayRep(:${*}:) (MinArgs=1, MaxArgs=2, Inline=Yes)
    ADR = Adr(:\$[1]:) (NumArgs=1, Inline=Yes)
    SIZEOF = Sizeof(:\$[1]:) (NumArgs=1, Inline=Yes)
    NUM_LOADED_FILES = NumLoadedFiles(::) (NumArgs=0)
    NUM_LOADED_PROG_FILES = NumLoadedProgFiles(::) (NumArgs=0)
    MEM_SIZE_IP_ALL = MemSizeIpInstAll(::) (NumArgs=0)
    MEM_SIZE_IP_LIB = MemSizeIpInst(::) (NumArgs=0)
    MEM_SIZE_SHLIB = MemSizeShLib(::) (NumArgs=0)
    MEM_SIZE_FILE = MemSizeFile(:$[1]:) (MinArgs=0, MaxArgs=1)
    MEM_SIZE_IP_STACK_SPACE = MemStackSpace(::) (NumArgs=0)
  AxesSpec:
    AxisRef = $\s*=\s*AC (Mode=3)
    AxisRef = $\s*=\s*IC (Mode=4)
  PVMacros:
    SBLOF (ArrayDims=0, Group=500)
      CALL = #call->forbid_stepping = 1; (Inline=Yes)
    SBLON (ArrayDims=0, Group=500)
      CALL = #call->forbid_stepping = 0; (Inline=Yes)
    DISPLOF (ArrayDims=0, Group=500)
      CALL = #call->forbid_display = 1; (Inline=Yes)
    DISPLON (ArrayDims=0, Group=500)
      CALL = #call->forbid_display = 0; (Inline=Yes)
    RDISABLE (ArrayDims=0, Group=500)
      CALL = @#job->sa.keep_alive = 1;
        @#thread.sa_keep_alive = 1; (Inline=Yes)
    P_SUBPAR $P_SUBPAR (ArrayDims=1, Group=500)
      GET = return ArgNumIsDefined(:$[1]:);
    P_STACK $P_STACK:
      GET = return UserCallDepth(::);
  FubTemplates:
    StdFubTemplate (IsDefault=Yes, Inline=Yes)
      Arg (ref=FUBINST, DataType=FLOAT)
      Arg (ref=FUBERRLEV, DataType=FLOAT)
      Arg (ref=PATHSYNCH, DataType=FLOAT)
      Arg (ref=BLOCKING, DataType=FLOAT)
  SynchActions:
    SABlocks:
      default (IsDefault=Yes)
        cyclic (Inline=Yes)
          Arg (ref=ACTIONS, DataType=STATEMENTS)
          Arg (ref=ID, DataType=FLOAT, DefaultInt=-1, MinCount=0, MaxCount=1)
      whenever:
        cyclic (Inline=Yes)
          Arg (ref=COND, DataType=FLOAT)
          Arg (ref=ACTIONS, DataType=STATEMENTS)
          Arg (ref=ID, DataType=FLOAT, DefaultInt=-1, MinCount=0, MaxCount=1)
      when:
        cyclic (Inline=Yes)
          Arg (ref=COND, DataType=FLOAT)
          Arg (ref=ACTIONS, DataType=STATEMENTS)
          Arg (ref=ID, DataType=FLOAT, DefaultInt=-1, MinCount=0, MaxCount=1)
      every:
        cyclic (Inline=Yes)
          Arg (ref=COND, DataType=FLOAT)
          Arg (ref=ACTIONS, DataType=STATEMENTS)
          Arg (ref=ID, DataType=FLOAT, DefaultInt=-1, MinCount=0, MaxCount=1)
      from:
        cyclic (Inline=Yes)
          Arg (ref=COND, DataType=FLOAT)
          Arg (ref=ACTIONS, DataType=STATEMENTS)
          Arg (ref=ID, DataType=FLOAT, DefaultInt=-1, MinCount=0, MaxCount=1)
    NonModalActivation:
      Start = @#thread.sa_last_keep_alive = 1;
        ActivateCyclicGroup(:-1:);
      Stop = WaitStopCyclicGroups(:(:-1:):);
  ParserData (NestedComments=Yes, DefaultCaseSensitive=No, CommentsSpanLines=No, SubDeclsLocalToFile=Yes, ProgDeclsLocalToFile=Yes, AllowUnprefixedFileCalls=Yes, AllowUnprefixedSubCalls=Yes, LocalVarScopeForMainProg=No, FileScopeVarsVisibleInSub=Yes, MainPrgReturnAtNextMainPrgHdr=Yes, AllowVarReadBeforeAssign=No, AllowArrayRefWithoutIndex=Yes, AllowNamedFnArgs=Yes, AllowBuiltinFnArgsOutOfSequence=Yes, AllowBuiltInProcCallWithoutBrackets=Yes, AllowBuiltInFnCallWithoutBrackets=No, AllowPLCFnCallWithoutBrackets=No, AllowStructMemberAutoDereference=Yes, AllowVariableAutoDereference=Yes, EnableStringCharacterIndexing=Yes, AllowIgnoredExtraSubArgs=Yes, OnMacroRedefinition=Error, CheckFileTimestampBeforeCalls=Yes)
    TKG_END_OF_LINE = \n (IsPattern=No)
    TKG_LINE_CONTINUE = \ (IsPattern=No, FileXLInvalid=Yes)
    TKG_LINE_BREAK = @@
    TKG_OPEN_COMMENT = ;
    TKG_CLOSE_COMMENT
    TKG_TRUE = TRUE:\W (IsPattern=Yes)
    TKG_FALSE = FALSE:\W (IsPattern=Yes)
    TKG_PAREVAL_MODAL_ID = ID:[\s=] (FileXLInvalid=Yes, IsPattern=Yes)
    TKG_MACRO_DEFINE_GLOBAL = define\s+ip_global:\s (IsPattern=Yes, FollowedBy=TKG_MACRO_NAME)
    TKG_MACRO_DEFINE = define\s+local:\s|define:\s (IsPattern=Yes, FollowedBy=TKG_MACRO_NAME)
    TKG_MACRO_UNDEFINE = undefine:\s (IsPattern=Yes, FollowedBy=TKG_MACRO_NAME)
    TKG_MACRO_AS = as:[\s\n] (IsPattern=Yes, FollowedBy=TKG_MACRO_TEXT)
    TKG_PROG_START = %:[^L] (IsPattern=Yes, CaseSensitive=Yes, FollowedBy=TKG_PROG_NAME)
    TKG_PROG_NAME = [\w\d]+ (IsPattern=Yes, Restricted=Yes)
    TKG_SET_MODAL_SUB = MCALL:\W (FileXLInvalid=Yes, IsPattern=Yes)
    TKG_INDIR_PROG_CALL = CALL:\s (IsPattern=Yes)
    TKG_INDIR_PROG_BLOCK = BLOCK:\s (FileXLInvalid=Yes, IsPattern=Yes)
    TKG_PROC_START = PROC:\s (FileXLInvalid=Yes, IsPattern=Yes, FollowedBy=TKG_PROC_NAME)
    TKG_PROC_NAME = \w[\w\d]+ (IsPattern=Yes, Restricted=Yes)
    TKG_ARG_PASSBYREF = VAR:\s (IsPattern=Yes)
    TKG_SUBPROG_PROTO = INTERN:\s (IsPattern=Yes, FollowedBy=TKG_SUBPROG_NAME)
    TKG_SUBPROG_START = SUB\s|%:L (FileXLInvalid=Yes, IsPattern=Yes, CaseSensitive=Yes, FollowedBy=TKG_SUBPROG_NAME)
    TKG_SUBPROG_NAME = \w[\w\d]+ (IsPattern=Yes, Restricted=Yes)
    TKG_EXTERN = EXTERN:\s (IsPattern=Yes, FollowedBy=TKG_PROG_FILE_NAME)
    TKG_PROG_FILE_NAME = [\^#&@']?[\w\d\./\:]+ (IsPattern=Yes, Restricted=Yes)
    TKG_PV_DECL = def:\s (IsPattern=Yes)
    TKG_PV_UNDECL = ~def:\s (IsPattern=Yes)
    TKG_VAR_RETAIN = retain:\s (IsPattern=Yes)
    TKG_VARSCOPE_IP_LOCAL = local:[\s\n] (IsPattern=Yes)
    TKG_VARSCOPE_IP_GLOBAL = ip_global:[\s\n] (IsPattern=Yes)
    TKG_VARSCOPE_NC_GLOBAL = nc_global:[\s\n] (IsPattern=Yes)
    TKG_VARSCOPE_PLC_GLOBAL = plc_global:[\s\n] (IsPattern=Yes)
    TKG_VARSYNCH_IP = ip_synch:\s (IsPattern=Yes)
    TKG_VARSYNCH_PATH = path_synch:\s (IsPattern=Yes)
    TKG_PAREVAL_DO = do:\s (FileXLInvalid=Yes, IsPattern=Yes)
    TKG_GOTOF = gotof:\s (FileXLInvalid=Yes, IsPattern=Yes, OptFollowedBy=TKG_GOTO_DEST)
    TKG_GOTOB = gotob:\s (FileXLInvalid=Yes, IsPattern=Yes, OptFollowedBy=TKG_GOTO_DEST)
    TKG_GOTO = goto:\s (FileXLInvalid=Yes, IsPattern=Yes, OptFollowedBy=TKG_GOTO_DEST)
    TKG_GOTO_DEST = \w[\w\d]* (IsPattern=Yes, Restricted=Yes)
    TKG_ARITH_BINARY_INT_DIVIDE = DIV:[\s(] (IsPattern=Yes)
    TKG_ARITH_BINARY_MODULO = MOD:[\s(] (IsPattern=Yes)
    TKG_FOR = FOR:\s (FileXLInvalid=Yes, IsPattern=Yes)
    TKG_ENDFOR = ENDFOR:[\s\n] (FileXLInvalid=Yes, IsPattern=Yes)
    TKG_FORTO = TO:\W (IsPattern=Yes)
    TKG_DO = repeat:[\s\n] (FileXLInvalid=Yes, IsPattern=Yes)
    TKG_ENDDO_UNTIL = until:[\s(] (FileXLInvalid=Yes, IsPattern=Yes)
    TKG_LOGICAL_UNARY_NOT = not:\W (IsPattern=Yes)
    TKG_SUPPRESS_SINGLE_STEP = NOHALT
    TKG_NC_BLOCK_PREFIX = N:[\s\d] (IsPattern=Yes)
    TKG_LOGICAL_HP_BINARY_AND = and:\W (IsPattern=Yes)
    TKG_LOGICAL_HP_BINARY_OR = or:\W (IsPattern=Yes)
    TKG_LOGICAL_HP_BINARY_XOR = xor:\W (IsPattern=Yes)
    TKG_BITWISE_BINARY_AND = b_and:\W (IsPattern=Yes)
    TKG_BITWISE_BINARY_OR = b_or:\W (IsPattern=Yes)
    TKG_BITWISE_BINARY_XOR = b_xor:\W (IsPattern=Yes)
    TKG_BITWISE_UNARY_COMPLEMENT = b_not:\W (IsPattern=Yes)
    TKG_IF = if:\W (FileXLInvalid=Yes, IsPattern=Yes)
    TKG_THEN = then:\W (FileXLInvalid=Yes, IsPattern=Yes)
    TKG_BLOCK_ELSE = else:\W (FileXLInvalid=Yes, IsPattern=Yes)
    TKG_BLOCK_ENDIF = endif:\W (FileXLInvalid=Yes, IsPattern=Yes)
    TKG_SWITCH = case:\W (FileXLInvalid=Yes, IsPattern=Yes)
    TKG_SWITCH_OF = of:\W (FileXLInvalid=Yes, IsPattern=Yes)
    TKG_SWITCH_DEFAULT = default:\W (FileXLInvalid=Yes, IsPattern=Yes)
    TKG_WHILE = while:\W (FileXLInvalid=Yes, IsPattern=Yes)
    TKG_ENDWHILE = endwhile (FileXLInvalid=Yes)
    TKG_FOREVER = loop:\W (FileXLInvalid=Yes, IsPattern=Yes)
    TKG_ENDFOREVER = endloop:\W (FileXLInvalid=Yes, IsPattern=Yes)
    TKG_LABEL_DEF = \w:\:|\w[\w\d]+:\: (IsPattern=Yes, FollowedBy=TKG_LABEL_SUFFIX)
    TKG_LABEL_SUFFIX = : (Restricted=Yes)
    TKG_MACRO_TEXT = . (Restricted=Yes, IsPattern=Yes)
    TKG_MACRO_NAME = [$\w][$\w\d(]+ (Restricted=Yes, IsPattern=Yes)
    TKG_PRIM_TYPE (IsPattern=Yes)
    TKG_OPEN_BRACKET = (
    TKG_CLOSE_BRACKET = )
    TKG_OPEN_INDEXBRACKET = [
    TKG_CLOSE_INDEXBRACKET = ]
    TKG_COMMA = ,
    TKG_DOT = \.:\w (IsPattern=Yes, FollowedBy=TKG_STRUCT_MEMBER_REF)
    TKG_STRUCT_MEMBER_REF = \w|\w[\w\d]+ (IsPattern=Yes, Restricted=Yes)
    TKG_PARAM_PREFIX = R:[\[\d]|$[RP]:[\[\d]|M[WLF]:[\[\d]|EX[WLBF]:[\[\d] (IsPattern=Yes)
    TKG_SUBRANGE = ..
    TKG_NUMBER = \d+\.\d+|\d+\.:[^\.] (IsPattern=Yes)
    TKG_INTEGER = \d+ (IsPattern=Yes)
    TKG_FRACTION = \.\d+ (IsPattern=Yes)
    TKG_NUMBER_EXP = EX:[\s\d\+\-\.] (IsPattern=Yes)
    TKG_STRING_CONCAT = <<
    TKG_COMP_BINARY_GREATER_THAN_OR_EQ = >=
    TKG_COMP_BINARY_LESS_THAN_OR_EQ = <=
    TKG_COMP_BINARY_EQUAL_TO = ==
    TKG_COMP_BINARY_NOT_EQUAL_TO = <>
    TKG_COMP_BINARY_GREATER_THAN = >
    TKG_COMP_BINARY_LESS_THAN = <
    TKG_ASSIGN_INCR = =ic:( (IsPattern=Yes)
    TKG_ASSIGN_EQ = =
    TKG_ARITH_BINARY_PLUS = +
    TKG_ARITH_BINARY_MINUS = -
    TKG_ARITH_BINARY_MULTIPLY = *
    TKG_ARITH_BINARY_DIVIDE = /
    TKG_SUBCALL_REPEAT_PREFIX = P:[\s\d] (IsPattern=Yes, FollowedBy=TKG_INTEGER)
    TKG_PV_DECL_REF = \w[\w\d\.\:\*]* (IsPattern=Yes, Restricted=Yes)
    TKG_G_CODE_PREFIX = G:[\s\d] (IsPattern=Yes)
    TKG_M_CODE_PREFIX = M:[\s\d(] (IsPattern=Yes)
    TKG_FUB_DECL = fub\s (IsPattern=Yes)
    TKG_FUB_ERR_LEV_1 = error_level_1:\s (IsPattern=Yes)
    TKG_FUB_ERR_LEV_2 = error_level_2:\s (IsPattern=Yes)
    TKG_FUB_ERR_LEV_3 = error_level_3:\s (IsPattern=Yes)
    TKG_FUB_ERR_LEV_4 = error_level_4:\s (IsPattern=Yes)
    TKG_FUB_BLOCKING = blocking:[\s\n] (IsPattern=Yes)
    TKG_FUB_NON_BLOCKING = non_blocking:\s (IsPattern=Yes)
    TKG_IEC_TYPED_VALUE = #[\w\d]+:[^\w\d\:] (IsPattern=Yes)
    TKG_REFERENCE = ref:[\s\n]|reference:[\s\n] (IsPattern=Yes, FollowedBy=TKG_IEC_TO)
    TKG_IEC_TO = to:[\s\n] (IsPattern=Yes, Restricted=Yes)
    TKG_ACCESS = ACCESS:[\s\n] (IsPattern=Yes)
    TKG_BINARY_LITERAL_START = 'B:[01_] (FollowedBy=TKG_BINARY_LITERAL_BODY, IsPattern=Yes)
    TKG_BINARY_LITERAL_BODY = [01_]+' (Restricted=Yes, IsPattern=Yes)
    TKG_HEX_LITERAL_START = 'H:[\dA-F_] (FollowedBy=TKG_HEX_LITERAL_BODY, IsPattern=Yes)
    TKG_HEX_LITERAL_BODY = [\dA-F_]+' (Restricted=Yes, IsPattern=Yes)
    TKG_WORD = \w|\w[\w\d\./]+|\./\w|\./\w[\w\d\./]+|[\^#][\w\d]+\:[\w\d\./]+ (IsPattern=Yes)
  StringChars (AsciiStringStart=", AsciiStringEnd=", UTF16StringStart=W", UTF16StringEnd=")
    EscapeSeq (Search=$N, ReplaceValue=10)
    EscapeSeq (Search=$L, ReplaceValue=10)
    EscapeSeq (Search=$P, ReplaceValue=12)
    EscapeSeq (Search=$R, ReplaceValue=13)
    EscapeSeq (Search=$T, ReplaceValue=9)
    EscapeSeq (Search=$Q, ReplaceStr=")
    EscapeSeq (Search=$', ReplaceStr=')
    EscapeSeq (Search=$", ReplaceStr=")
    EscapeSeq (Search=$[\dA-Fa-f]+, IsPattern=Yes, ReplaceEncodingBase=16)
    EscapeSeq (Search=$$, ReplaceStr=$)
    EscapeSeq (Search=$, ReplaceStr=)
```

### Data object Logical/MotionHandling/Interpreter/GmcIpConfig/gmcipcsm (Cnc, version 2.47.4)

#### gmcipcsm.cnc
```
Root (LangModule=ailgcode, Version=1.0)
  Constants:
    NumAxes = 15 (Type=INT)
  Preprocess:
    PP_RULE_STOPRE (Search=STOPRE, Replace=G172)
    PP_RULE_CIP (Search=CIP:\W, Replace=G102, IsPattern=Yes)
  Types:
    RotationAngleSpecifier (type=ENUM, EnumType=REGEXP, Value6=H)
    RadiusSpecifier (type=ENUM, EnumType=REGEXP, Value1=R\s*=, Value2=CR\s*=)
    InterpolParam (type=ENUM, EnumType=REGEXP, Value0=I, Value1=J, Value2=K, Value100=G161\s*I, Value101=G161\s*J, Value102=G161\s*K, Value200=G162\s*I, Value201=G162\s*J, Value202=G162\s*K, Value0300=I\s*=\s*AC, Value0301=J\s*=\s*AC, Value0302=K\s*=\s*AC, Value0400=I\s*=\s*IC, Value0401=J\s*=\s*IC, Value0402=K\s*=\s*IC)
    CirclePointParam (type=ENUM, EnumType=REGEXP, Value0=I1\s*=, Value1=J1\s*=, Value2=K1\s*=, Value100=G161\s*I1\s*=, Value101=G161\s*J1\s*=, Value102=G161\s*K1\s*=, Value200=G162\s*I1\s*=, Value201=G162\s*J1\s*=, Value202=G162\s*K1\s*=, Value0300=I1\s*=\s*AC, Value0301=J1\s*=\s*AC, Value0302=K1\s*=\s*AC, Value0400=I1\s*=\s*IC, Value0401=J1\s*=\s*IC, Value0402=K1\s*=\s*IC)
    RPYAngleName (type=ENUM, EnumType=REGEXP, Value1=ROLL, Value0=PITCH, Value2=YAW)
    EulerAngleName (type=ENUM, EnumType=REGEXP, Value3=PHI, Value4=THETA, Value5=PSI)
    RotaryVectorName (type=ENUM, EnumType=REGEXP, Value0=P\s*=, Value1=Q\s*=, Value2=R\s*=)
    DwellTime (type=FLOAT)
    RParamIndex (type=INT, MinValue=0, MaxValue=999)
    EXParamIndex (type=INT, MinValue=0, MaxValue=99)
    MParamIndex (type=INT, MinValue=0, MaxValue=99)
    Byte (type=INT, MinValue=0, MaxValue=255)
    Word (type=INT, MinValue=-32768, MaxValue=32767)
    Long (type=INT)
    AxisAccelPercentage (type=FLOAT, MinValue=0.0000001, MaxValue=100)
  PVMacros:
    SAVE (ArrayDims=0, Group=500)
      CALL = Info(:id:52101, msg:"Save Modal GCode State NOT SUPPORTED YET":);
  SysVars:
    P_F $P_F:
      GET = return @%_CNC.v_ncprog;
    P_GG $P_GG:
      GET = return @%_CNC.typ_ncblock;
    LIM_PATH_V $LIM_PATH_V:
      GET = return %_CNC.lim_path_v;
      SET:
        ARG (ref=EXPR, DataType=FLOAT)
    LIM_PATH_ACC_P $LIM_PATH_ACC_P:
      GET = return %_CNC.lim_path_acc_p;
      SET:
        ARG (ref=EXPR, DataType=FLOAT)
    LIM_PATH_ACC_N $LIM_PATH_ACC_N:
      GET = return %_CNC.lim_path_acc_n;
      SET:
        ARG (ref=EXPR, DataType=FLOAT)
    S_JUMP_T $S_JUMP_T:
      GET = return %_CNC.s_jump_t;
      SET:
        ARG (ref=EXPR, DataType=FLOAT)
    RADIUS_ERR $RADIUS_ERR:
      GET = return %_CNC.radius_err;
      SET:
        ARG (ref=EXPR, DataType=FLOAT)
    V_JUMP_T $V_JUMP_T:
      GET = return %_CNC.v_jump_t;
      SET:
        ARG (ref=EXPR, DataType=FLOAT)
    LIM_AX_ACC $LIM_AX_ACC (ArrayDims=1)
      GET = return %_AX.a_max_ncdy[$[1]];
      SET:
        ARG (ref=EXPR, DataType=FLOAT)
    LIM_ACC ACC (ArrayDims=1)
      GET = return %_AX.a_max_ncdy[$[1]] / %_AX.a_max[$[1]] * 100.0;
      SET:
        ARG (ref=EXPR, DataType=AxisAccelPercentage)
    LIM_AX_V $LIM_AX_V (ArrayDims=1)
      GET = return %_AX.v_max_ncdy[$[1]];
      SET:
        ARG (ref=EXPR, DataType=FLOAT)
    AX_A_JUMP $AX_A_JUMP (ArrayDims=1)
      GET = return %_AX.a_jump_ncdy[$[1]];
      SET:
        ARG (ref=EXPR, DataType=FLOAT)
    AX_V_JUMP $AX_V_JUMP (ArrayDims=1)
      GET = return %_AX.v_jump_ncdy[$[1]];
      SET:
        ARG (ref=EXPR, DataType=FLOAT)
    AX_T_INPOS $AX_T_INPOS (ArrayDims=1)
      GET = return %_AX.t_inpos[$[1]];
    AX_T_IN_POS $AX_T_IN_POS (ArrayDims=1)
      GET = return %_AX.t_inpos[$[1]];
    AX_T_JOLT $AX_T_JOLT (ArrayDims=1)
      GET = return %_AX.t_jolt_ax[$[1]];
    PATH_T_JOLT $PATH_T_JOLT:
      GET = return %_CNC.path_t_jolt;
    LIM_PATH_ACC_P_INI $LIM_PATH_ACC_P_INI:
      GET = return %_CNC.lim_path_acc_p_ini;
    LIM_PATH_ACC_N_INI $LIM_PATH_ACC_N_INI:
      GET = return %_CNC.lim_path_acc_n_ini;
    AA_IM $AA_IM (ArrayDims=1)
      GET = return @%_AX.set_pos_mcs[$[1]];
    AA_IW $AA_IW (ArrayDims=1)
      GET = return @%_AX.set_pos[$[1]];
    P_SIM $P_SIM (ArrayDims=1)
      GET = return %_AX.sim_status[$[1]];
    MA_MAX_AX_ACCEL $MA_MAX_AX_ACCEL (ArrayDims=1)
      GET = return %_AX.a_max[$[1]];
    MA_MAX_AX_VELO $MA_MAX_AX_VELO (ArrayDims=1)
      GET = return %_AX.v_max[$[1]];
    MA_MAX_AX_JERK $MA_MAX_AX_JERK (ArrayDims=1)
      GET = return %_AX.jerk_max[$[1]];
    MA_POSCTRL_GAIN $MA_POSCTRL_GAIN (ArrayDims=1)
      GET = return %_AX.servo_gain[$[1]];
    MA_REFP_SET_POS $MA_REFP_SET_POS (ArrayDims=1)
      GET = return %_AX.home_pos[$[1]];
    MA_POS_LIMIT_PLUS $MA_POS_LIMIT_PLUS (ArrayDims=1)
      GET = return %_AX.pos_sw_end[$[1]];
    MA_POS_LIMIT_MINUS $MA_POS_LIMIT_MINUS (ArrayDims=1)
      GET = return %_AX.neg_sw_end[$[1]];
  Parameters:
    R (IndexType=RParamIndex, ValueType=FLOAT)
      ARG (ref=EXPR, DataType=RParamIndex)
    QUOTED (QuotedName=$R, Synchronous=Yes, IndexType=RParamIndex, ValueType=FLOAT)
      ARG (ref=EXPR, DataType=RParamIndex)
    QUOTED (QuotedName=$P, Synchronous=Yes, IndexType=RParamIndex, ValueType=FLOAT)
      ARG (ref=EXPR, DataType=RParamIndex)
    EXB (IndexType=EXParamIndex, ValueType=Byte)
      ARG (ref=EXPR, DataType=EXParamIndex)
    EXW (IndexType=EXParamIndex, ValueType=Word)
      ARG (ref=EXPR, DataType=EXParamIndex)
    EXL (IndexType=EXParamIndex, ValueType=Long)
      ARG (ref=EXPR, DataType=EXParamIndex)
    EXF (IndexType=EXFParamIndex, ValueType=FLOAT)
      ARG (ref=EXPR, DataType=EXFParamIndex)
    MW (Synchronous=Yes, IndexType=MParamIndex, ValueType=Word)
      ARG (ref=EXPR, DataType=MParamIndex)
    ML (Synchronous=Yes, IndexType=MParamIndex, ValueType=Long)
      ARG (ref=EXPR, DataType=MParamIndex)
    MF (Synchronous=Yes, IndexType=MParamIndex, ValueType=FLOAT)
      ARG (ref=EXPR, DataType=MParamIndex)
  MCodes:
    M17 = 17 (Group=41, Alias=RET:[^\d\w\(], Eval=Early, Inline=Yes, AliasIsPattern=Yes)
      ARG (ref=VALUE, DataType=FLOAT, RequireLiteral=Yes)
    M17_1 = 17.1 (Group=41, Alias=CONDRET, Eval=Early, Inline=Yes)
      ARG (ref=VALUE, DataType=FLOAT, RequireLiteral=Yes)
```

### Data object Logical/MotionHandling/Interpreter/GmcIpConfig/gmcipcfg (Cnc, version 2.47.4)

#### gmcipcfg.cnc
```
CONFIG:
  LANG_INCLUDE gmcipmxd (LangName=IEC-ST, DataObject=Yes, IfNotExist=Error, Scope=NC_GLOBAL, RequireFnIgnore=MXConvertOrient)
  XML_INCLUDE gmcipvar (IfNotExist=Warn)
  XML_INCLUDE gmcipfun (IfNotExist=Warn)
  XML_INCLUDE gmcipfub (IfNotExist=Warn)
  MPQUEUE (NumPackets=200, LookaheadMinBlocks=5, LookaheadMaxBlocks=20, LookaheadMode=any, MaxPathJobs=256)
  MONITOR (MaxPathStackEvents=1024)
  MPLOG (MaxBuffers=10, MinBuffers=4, EarlyCircleBufferLookahead=2, DefaultBufferSize=131072, TaskCycleDelay=1, FileDevice=mplog*, MaxLogFiles=20, MaxLogFileSize=1048576, CopyLineTextMaxChars=80)
  AXES (StandardCNCAxes=Yes)
  FUBOutputs:
    FUBOutput PLCOpen:
      ERROR (condition=$Error == 1)
      BUSY (condition=$Busy == 1)
    FUBOutput BuR:
      ERROR (condition=$status != 65535 && $status != 0)
      BUSY (condition=$status == 65535)
  FUNCTIONS:
    FUNC LEN (DeclareName=__LEN, AlwaysDeclare=Yes, RetType=INT)
      ARG IN (Type=STRING)
    FUNC LEFT (DeclareName=__LEFT, AlwaysDeclare=Yes, RetType=STRING, RetRef=Yes)
      ARG IN (Type=STRING)
      ARG L (Type=INT)
    FUNC RIGHT (DeclareName=__RIGHT, AlwaysDeclare=Yes, RetType=STRING, RetRef=Yes)
      ARG IN (Type=STRING)
      ARG L (Type=INT)
    FUNC MID (DeclareName=__MID, AlwaysDeclare=Yes, RetType=STRING, RetRef=Yes)
      ARG IN (Type=STRING)
      ARG L (Type=INT)
      ARG P (Type=INT)
    FUNC CONCAT (DeclareName=__CONCAT, AlwaysDeclare=Yes, RetType=STRING, RetRef=Yes)
      ARG IN1 (Type=STRING)
      ARG IN2 (Type=STRING)
    FUNC INSERT (DeclareName=__INSERT, AlwaysDeclare=Yes, RetType=STRING, RetRef=Yes)
      ARG IN1 (Type=STRING)
      ARG IN2 (Type=STRING)
      ARG P (Type=INT)
    FUNC DELETE (DeclareName=__DELETE, AlwaysDeclare=Yes, RetType=STRING, RetRef=Yes)
      ARG IN (Type=STRING)
      ARG L (Type=INT)
      ARG P (Type=INT)
    FUNC REPLACE (DeclareName=__REPLACE, AlwaysDeclare=Yes, RetType=STRING, RetRef=Yes)
      ARG IN1 (Type=STRING)
      ARG IN2 (Type=STRING)
      ARG L (Type=INT)
      ARG P (Type=INT)
    FUNC FIND (DeclareName=__FIND, AlwaysDeclare=Yes, RetType=INT)
      ARG IN1 (Type=STRING)
      ARG IN2 (Type=STRING)
  XML_INCLUDE gmcipuc (IfNotExist=Warn)
```

### Data object Logical/MotionHandling/Interpreter/GmcIpConfig/gmcipiec (Cnc, version 2.47.4)

#### gmcipiec.cnc
```
Root (LangModule=ailgcode, Version=1.0)
  AxesSpec
  PrimTypes (PatternSuffix=:[^\d\w$#])
    BOOL (BRType=BOOL)
    STRING (BRType=STRING)
    WSTRING (BRType=WSTRING)
    TIME (BRType=TIME)
    SINT (BRType=SINT)
    INT (BRType=INT)
    DINT (BRType=DINT)
    USINT (BRType=USINT)
    UINT (BRType=UINT)
    UDINT (BRType=UDINT)
    REAL (BRType=REAL)
    LREAL (BRType=LREAL)
    DATE (BRType=DATE)
    DATE_AND_TIME (BRType=DATE_AND_TIME)
    DT (BRType=DT)
    TIME_OF_DAY (BRType=TIME_OF_DAY)
    TOD (BRType=TIME_OF_DAY)
    BYTE (BRType=BYTE)
    WORD (BRType=WORD)
    DWORD (BRType=DWORD)
  BuiltInProcs:
    SetCyclicId = #job->group_id = $[1]; (MinArgs=1, MaxArgs=1, Eval=Early)
    WaitForCyclic = if ( Defined(:$[1]:) ) 
        WaitForCyclicGroups(:${*}:);  
      else
        WaitForCyclicJob(:#last_job_id:);
      endif (MinArgs=0, MaxArgs=*)
    REPORT (MinArgs=2, MaxArgs=2)
      Arg (ref=id, DataType=INT)
      Arg (ref=msg, DataType=STRING)
    WARN (MinArgs=2, MaxArgs=2)
      Arg (ref=id, DataType=INT)
      Arg (ref=msg, DataType=STRING)
    HALT (MinArgs=2, MaxArgs=2)
      Arg (ref=id, DataType=INT)
      Arg (ref=msg, DataType=STRING)
    ERROR (MinArgs=2, MaxArgs=2)
      Arg (ref=id, DataType=INT)
      Arg (ref=msg, DataType=STRING)
    LOADBG (MinArgs=1, MaxArgs=1)
      Arg (ref=filename, DataType=STRING)
    LOAD (MinArgs=1, MaxArgs=1)
      Arg (ref=filename, DataType=STRING)
    UNLOAD (MinArgs=1, MaxArgs=1)
      Arg (ref=filename, DataType=STRING)
    EXEC (MinArgs=1, MaxArgs=3)
      Arg (ref=filename, DataType=STRING)
      Arg (ref=arguments, DataType=ANY_DATA)
      Arg (ref=langId, DataType=INT)
    EVAL = local $file_id;
      $file_id = LoadProgString(:$[1], $[2]:);
      WaitForLoadProg(:$file_id:);
      ExecProg(:$file_id:);
      UnloadProg(:$file_id:); (MinArgs=1, MaxArgs=2)
    PUSH_PACKET = PushPacket(::);
    PUSH_PACKET_CMD (MinArgs=1, MaxArgs=2)
      Arg (ref=cmd, DataType=INT)
      Arg (ref=data, DataType=ANY_DATA)
    DISPATCH_AND_WAIT (MinArgs=1, MaxArgs=1)
      Arg (ref=cmd, DataType=INT)
    START_PACKET_LIST = #inhibit_mp_list_dispatch = 1;
    END_PACKET_LIST = #inhibit_mp_list_dispatch = 0;
    LOG_INFO (MinArgs=1, MaxArgs=1)
      Arg (ref=msg, DataType=STRING)
    SET_BLOCK_NUMBER = SetCurBlockNr(:$[1]:); (MinArgs=1, MaxArgs=1)
    SBLOF_PATH = #next_motion.Command = MPCMD_SBL_PATH_INHIBIT;
      PushPacket(::);
    SBLON_PATH = #next_motion.Command = MPCMD_SBL_PATH_RELEASE;
      PushPacket(::);
  BuiltInFns:
    ABS = Abs(:$[1]:) (ReturnType=ANY_NUM, ArgType1=ANY_NUM, Inline=Yes)
    SIN = RSin(:$[1]:) (ReturnType=ANY_REAL, ArgType1=ANY_REAL, Inline=Yes)
    COS = RCos(:$[1]:) (ReturnType=ANY_REAL, ArgType1=ANY_REAL, Inline=Yes)
    TAN = RTan(:$[1]:) (ReturnType=ANY_REAL, ArgType1=ANY_REAL, Inline=Yes)
    ASIN = RASin(:$[1]:) (ReturnType=ANY_REAL, ArgType1=ANY_REAL, Inline=Yes)
    ACOS = RACos(:$[1]:) (ReturnType=ANY_REAL, ArgType1=ANY_REAL, Inline=Yes)
    ATAN = RATan(:$[1]:) (ReturnType=ANY_REAL, ArgType1=ANY_REAL, Inline=Yes)
    SQRT = Sqrt(:$[1]:) (ReturnType=ANY_REAL, ArgType1=ANY_REAL, Inline=Yes)
    LN = Ln(:$[1]:) (ReturnType=ANY_REAL, ArgType1=ANY_REAL, Inline=Yes)
    EXP = Exp(:$[1]:) (ReturnType=ANY_REAL, ArgType1=ANY_REAL, Inline=Yes)
    LOG = Log(:$[1]:) (ReturnType=ANY_REAL, ArgType1=ANY_REAL, Inline=Yes)
    EXPT = Pow(:$[1],$[2]:) (ReturnType=ANY_REAL, ArgType1=ANY_REAL, ArgType2=ANY_NUM, Inline=Yes)
    TRUNC = ToInt(:Fix(:$[1]:):) (ReturnType=IEC_INT, ArgType1=FLOAT, Inline=Yes)
    ADR = Adr(:\$[1]:) (ReturnType=IEC_UDINT, ArgType1=ANY_DATA, Inline=Yes)
    REF = \$[1] (ReturnType=ANY_DATA, ArgType1=ANY_DATA, Inline=Yes)
    SIZEOF = Sizeof(:\$[1]:) (ReturnType=IEC_UINT, NumArgs=1, Inline=Yes)
    LIMIT (ReturnType=ANY_NUM, Inline=No)
      Arg (ref=MIN, DataType=ANY_NUM)
      Arg (ref=IN, DataType=ANY_NUM)
      Arg (ref=MAX, DataType=ANY_NUM)
    MIN (ReturnType=ANY_NUM, Inline=No)
      Arg (ref=IN1, DataType=ANY_NUM)
      Arg (ref=IN2, DataType=ANY_NUM)
    MAX (ReturnType=ANY_NUM, Inline=No)
      Arg (ref=IN1, DataType=ANY_NUM)
      Arg (ref=IN2, DataType=ANY_NUM)
    ROL = BitRotL(:$[1],$[2]:) (ReturnType=ANY_NUM, ArgType1=ANY_NUM, ArgType2=IEC_SINT)
    ROR = BitRotR(:$[1],$[2]:) (ReturnType=ANY_NUM, ArgType1=ANY_NUM, ArgType2=IEC_SINT)
    SHR = BitShR(:$[1],$[2]:) (ReturnType=ANY_NUM, ArgType1=ANY_NUM, ArgType2=IEC_SINT)
    SHL = BitShL(:$[1],$[2]:) (ReturnType=ANY_NUM, ArgType1=ANY_NUM, ArgType2=IEC_SINT)
    BIT_TST = AsBitTst(:$[1],$[2]:) (ReturnType=ANY_NUM, ArgType1=ANY_NUM, ArgType2=IEC_SINT)
    BIT_SET = AsBitSet(:$[1],$[2]:) (ReturnType=ANY_NUM, ArgType1=ANY_NUM, ArgType2=IEC_SINT)
    BIT_CLR = AsBitClr(:$[1],$[2]:) (ReturnType=ANY_NUM, ArgType1=ANY_NUM, ArgType2=IEC_SINT)
    TO_BOOL = ToBool(:$[1]:) (ReturnType=IEC_BOOL, ArgType1=ANY_DATA, Inline=Yes)
    TO_USINT = ToUInt(:$[1],1:) (ReturnType=IEC_USINT, ArgType1=ANY_DATA, Inline=Yes)
    TO_BYTE = ToUInt(:$[1],1:) (ReturnType=IEC_BYTE, ArgType1=ANY_DATA, Inline=Yes)
    TO_SINT = ToInt(:$[1],1:) (ReturnType=IEC_SINT, ArgType1=ANY_DATA, Inline=Yes)
    TO_UINT = ToUInt(:$[1],2:) (ReturnType=IEC_UINT, ArgType1=ANY_DATA, Inline=Yes)
    TO_WORD = ToUInt(:$[1],2:) (ReturnType=IEC_WORD, ArgType1=ANY_DATA, Inline=Yes)
    TO_INT = ToInt(:$[1],2:) (ReturnType=IEC_INT, ArgType1=ANY_DATA, Inline=Yes)
    TO_UDINT = ToUInt(:$[1]:) (ReturnType=IEC_UDINT, ArgType1=ANY_DATA, Inline=Yes)
    TO_DWORD = ToUInt(:$[1]:) (ReturnType=IEC_DWORD, ArgType1=ANY_DATA, Inline=Yes)
    TO_DINT = ToInt(:$[1]:) (ReturnType=IEC_DINT, ArgType1=ANY_DATA, Inline=Yes)
    TO_TIME = ToTime(:$[1]:) (ReturnType=IEC_TIME, ArgType1=ANY_DATA, Inline=Yes)
    TO_DT = ToDT(:$[1]:) (ReturnType=IEC_DT, ArgType1=ANY_DATA, Inline=Yes)
    TO_DATE_AND_TIME = ToDT(:$[1]:) (ReturnType=IEC_DT, ArgType1=ANY_DATA, Inline=Yes)
    TO_TOD = ToTOD(:$[1]:) (ReturnType=IEC_TOD, ArgType1=ANY_DATA, Inline=Yes)
    TO_TIME_OF_DAY = ToTOD(:$[1]:) (ReturnType=IEC_TOD, ArgType1=ANY_DATA, Inline=Yes)
    TO_DATE = ToDate(:$[1]:) (ReturnType=IEC_DATE, ArgType1=ANY_DATA, Inline=Yes)
    TO_REAL = ToFloat(:$[1]:) (ReturnType=IEC_REAL, ArgType1=ANY_DATA, Inline=Yes)
    TO_LREAL = ToLReal(:$[1]:) (ReturnType=IEC_LREAL, ArgType1=ANY_DATA, Inline=Yes)
    TO_STRING = ToString(:$[1]:) (ReturnType=IEC_STRING, ArgType1=ANY_DATA, Inline=Yes)
    TO_WSTRING = ToWString(:$[1]:) (ReturnType=IEC_WSTRING, ArgType1=ANY_DATA, Inline=Yes)
    USINT_TO_BOOL = ToBool(:$[1]:) (ReturnType=IEC_BOOL, ArgType1=IEC_USINT, Inline=Yes)
    SINT_TO_BOOL = ToBool(:$[1]:) (ReturnType=IEC_BOOL, ArgType1=IEC_SINT, Inline=Yes)
    UINT_TO_BOOL = ToBool(:$[1]:) (ReturnType=IEC_BOOL, ArgType1=IEC_UINT, Inline=Yes)
    INT_TO_BOOL = ToBool(:$[1]:) (ReturnType=IEC_BOOL, ArgType1=IEC_INT, Inline=Yes)
    UDINT_TO_BOOL = ToBool(:$[1]:) (ReturnType=IEC_BOOL, ArgType1=IEC_UDINT, Inline=Yes)
    DINT_TO_BOOL = ToBool(:$[1]:) (ReturnType=IEC_BOOL, ArgType1=IEC_DINT, Inline=Yes)
    REAL_TO_BOOL = ToBool(:$[1]:) (ReturnType=IEC_BOOL, ArgType1=IEC_REAL, Inline=Yes)
    LREAL_TO_BOOL = ToBool(:$[1]:) (ReturnType=IEC_BOOL, ArgType1=IEC_LREAL, Inline=Yes)
    TIME_TO_BOOL = ToBool(:$[1]:) (ReturnType=IEC_BOOL, ArgType1=IEC_TIME, Inline=Yes)
    DT_TO_BOOL = ToBool(:$[1]:) (ReturnType=IEC_BOOL, ArgType1=IEC_DT, Inline=Yes)
    TOD_TO_BOOL = ToBool(:$[1]:) (ReturnType=IEC_BOOL, ArgType1=IEC_TOD, Inline=Yes)
    BYTE_TO_BOOL = ToBool(:$[1]:) (ReturnType=IEC_BOOL, ArgType1=IEC_BYTE, Inline=Yes)
    WORD_TO_BOOL = ToBool(:$[1]:) (ReturnType=IEC_BOOL, ArgType1=IEC_WORD, Inline=Yes)
    DWORD_TO_BOOL = ToBool(:$[1]:) (ReturnType=IEC_BOOL, ArgType1=IEC_DWORD, Inline=Yes)
    BOOL_TO_USINT = ToUInt(:$[1],1:) (ReturnType=IEC_USINT, ArgType1=IEC_BOOL, Inline=Yes)
    SINT_TO_USINT = ToUInt(:$[1],1:) (ReturnType=IEC_USINT, ArgType1=IEC_SINT, Inline=Yes)
    UINT_TO_USINT = ToUInt(:$[1],1:) (ReturnType=IEC_USINT, ArgType1=IEC_UINT, Inline=Yes)
    INT_TO_USINT = ToUInt(:$[1],1:) (ReturnType=IEC_USINT, ArgType1=IEC_INT, Inline=Yes)
    UDINT_TO_USINT = ToUInt(:$[1],1:) (ReturnType=IEC_USINT, ArgType1=IEC_UDINT, Inline=Yes)
    DINT_TO_USINT = ToUInt(:$[1],1:) (ReturnType=IEC_USINT, ArgType1=IEC_DINT, Inline=Yes)
    REAL_TO_USINT = ToUInt(:$[1],1:) (ReturnType=IEC_USINT, ArgType1=IEC_REAL, Inline=Yes)
    LREAL_TO_USINT = ToUInt(:$[1],1:) (ReturnType=IEC_USINT, ArgType1=IEC_LREAL, Inline=Yes)
    BOOL_TO_SINT = ToInt(:$[1],1:) (ReturnType=IEC_SINT, ArgType1=IEC_BOOL, Inline=Yes)
    USINT_TO_SINT = ToInt(:$[1],1:) (ReturnType=IEC_SINT, ArgType1=IEC_USINT, Inline=Yes)
    UINT_TO_SINT = ToInt(:$[1],1:) (ReturnType=IEC_SINT, ArgType1=IEC_UINT, Inline=Yes)
    INT_TO_SINT = ToInt(:$[1],1:) (ReturnType=IEC_SINT, ArgType1=IEC_INT, Inline=Yes)
    UDINT_TO_SINT = ToInt(:$[1],1:) (ReturnType=IEC_SINT, ArgType1=IEC_UDINT, Inline=Yes)
    DINT_TO_SINT = ToInt(:$[1],1:) (ReturnType=IEC_SINT, ArgType1=IEC_DINT, Inline=Yes)
    REAL_TO_SINT = ToInt(:$[1],1:) (ReturnType=IEC_SINT, ArgType1=IEC_REAL, Inline=Yes)
    LREAL_TO_SINT = ToInt(:$[1],1:) (ReturnType=IEC_SINT, ArgType1=IEC_LREAL, Inline=Yes)
    BOOL_TO_UINT = ToUInt(:$[1],2:) (ReturnType=IEC_UINT, ArgType1=IEC_BOOL, Inline=Yes)
    SINT_TO_UINT = ToUInt(:$[1],2:) (ReturnType=IEC_UINT, ArgType1=IEC_SINT, Inline=Yes)
    USINT_TO_UINT = ToUInt(:$[1],2:) (ReturnType=IEC_UINT, ArgType1=IEC_USINT, Inline=Yes)
    INT_TO_UINT = ToUInt(:$[1],2:) (ReturnType=IEC_UINT, ArgType1=IEC_INT, Inline=Yes)
    UDINT_TO_UINT = ToUInt(:$[1],2:) (ReturnType=IEC_UINT, ArgType1=IEC_UDINT, Inline=Yes)
    DINT_TO_UINT = ToUInt(:$[1],2:) (ReturnType=IEC_UINT, ArgType1=IEC_DINT, Inline=Yes)
    REAL_TO_UINT = ToUInt(:$[1],2:) (ReturnType=IEC_UINT, ArgType1=IEC_REAL, Inline=Yes)
    LREAL_TO_UINT = ToUInt(:$[1],2:) (ReturnType=IEC_UINT, ArgType1=IEC_LREAL, Inline=Yes)
    BOOL_TO_INT = ToInt(:$[1],2:) (ReturnType=IEC_INT, ArgType1=IEC_BOOL, Inline=Yes)
    SINT_TO_INT = ToInt(:$[1],2:) (ReturnType=IEC_INT, ArgType1=IEC_SINT, Inline=Yes)
    USINT_TO_INT = ToInt(:$[1],2:) (ReturnType=IEC_INT, ArgType1=IEC_USINT, Inline=Yes)
    UINT_TO_INT = ToInt(:$[1],2:) (ReturnType=IEC_INT, ArgType1=IEC_UINT, Inline=Yes)
    UDINT_TO_INT = ToInt(:$[1],2:) (ReturnType=IEC_INT, ArgType1=IEC_UDINT, Inline=Yes)
    DINT_TO_INT = ToInt(:$[1],2:) (ReturnType=IEC_INT, ArgType1=IEC_DINT, Inline=Yes)
    REAL_TO_INT = ToInt(:$[1],2:) (ReturnType=IEC_INT, ArgType1=IEC_REAL, Inline=Yes)
    LREAL_TO_INT = ToInt(:$[1],2:) (ReturnType=IEC_INT, ArgType1=IEC_LREAL, Inline=Yes)
    BOOL_TO_UDINT = ToUInt(:$[1]:) (ReturnType=IEC_UDINT, ArgType1=IEC_BOOL, Inline=Yes)
    USINT_TO_UDINT = ToUInt(:$[1]:) (ReturnType=IEC_UDINT, ArgType1=IEC_USINT, Inline=Yes)
    SINT_TO_UDINT = ToUInt(:$[1]:) (ReturnType=IEC_UDINT, ArgType1=IEC_SINT, Inline=Yes)
    UINT_TO_UDINT = ToUInt(:$[1]:) (ReturnType=IEC_UDINT, ArgType1=IEC_UINT, Inline=Yes)
    INT_TO_UDINT = ToUInt(:$[1]:) (ReturnType=IEC_UDINT, ArgType1=IEC_INT, Inline=Yes)
    DINT_TO_UDINT = ToUInt(:$[1]:) (ReturnType=IEC_UDINT, ArgType1=IEC_DINT, Inline=Yes)
    REAL_TO_UDINT = ToUInt(:$[1]:) (ReturnType=IEC_UDINT, ArgType1=IEC_REAL, Inline=Yes)
    LREAL_TO_UDINT = ToUInt(:$[1]:) (ReturnType=IEC_UDINT, ArgType1=IEC_LREAL, Inline=Yes)
    TIME_TO_UDINT = ToUInt(:$[1]:) (ReturnType=IEC_UDINT, ArgType1=IEC_TIME, Inline=Yes)
    DT_TO_UDINT = ToUInt(:$[1]:) (ReturnType=IEC_UDINT, ArgType1=IEC_DT, Inline=Yes)
    BOOL_TO_DINT = ToInt(:$[1]:) (ReturnType=IEC_DINT, ArgType1=IEC_BOOL, Inline=Yes)
    USINT_TO_DINT = ToInt(:$[1]:) (ReturnType=IEC_DINT, ArgType1=IEC_USINT, Inline=Yes)
    SINT_TO_DINT = ToInt(:$[1]:) (ReturnType=IEC_DINT, ArgType1=IEC_SINT, Inline=Yes)
    UINT_TO_DINT = ToInt(:$[1]:) (ReturnType=IEC_DINT, ArgType1=IEC_UINT, Inline=Yes)
    INT_TO_DINT = ToInt(:$[1]:) (ReturnType=IEC_DINT, ArgType1=IEC_INT, Inline=Yes)
    UDINT_TO_DINT = ToInt(:$[1]:) (ReturnType=IEC_DINT, ArgType1=IEC_UDINT, Inline=Yes)
    REAL_TO_DINT = ToInt(:$[1]:) (ReturnType=IEC_DINT, ArgType1=IEC_REAL, Inline=Yes)
    LREAL_TO_DINT = ToInt(:$[1]:) (ReturnType=IEC_DINT, ArgType1=IEC_LREAL, Inline=Yes)
    TIME_TO_DINT = ToInt(:$[1]:) (ReturnType=IEC_DINT, ArgType1=IEC_TIME, Inline=Yes)
    DT_TO_DINT = ToInt(:$[1]:) (ReturnType=IEC_DINT, ArgType1=IEC_DT, Inline=Yes)
    BOOL_TO_TIME = ToTime(:$[1]:) (ReturnType=IEC_TIME, ArgType1=IEC_BOOL, Inline=Yes)
    DINT_TO_TIME = ToTime(:$[1]:) (ReturnType=IEC_TIME, ArgType1=IEC_DINT, Inline=Yes)
    UDINT_TO_TIME = ToTime(:$[1]:) (ReturnType=IEC_TIME, ArgType1=IEC_UDINT, Inline=Yes)
    BOOL_TO_DT = ToDT(:$[1]:) (ReturnType=IEC_DT, ArgType1=IEC_BOOL, Inline=Yes)
    DINT_TO_DT = ToDT(:$[1]:) (ReturnType=IEC_DT, ArgType1=IEC_DINT, Inline=Yes)
    UDINT_TO_DT = ToDT(:$[1]:) (ReturnType=IEC_DT, ArgType1=IEC_UDINT, Inline=Yes)
    BOOL_TO_REAL = ToFloat(:$[1]:) (ReturnType=IEC_REAL, ArgType1=IEC_BOOL, Inline=Yes)
    USINT_TO_REAL = ToFloat(:$[1]:) (ReturnType=IEC_REAL, ArgType1=IEC_USINT, Inline=Yes)
    SINT_TO_REAL = ToFloat(:$[1]:) (ReturnType=IEC_REAL, ArgType1=IEC_SINT, Inline=Yes)
    UINT_TO_REAL = ToFloat(:$[1]:) (ReturnType=IEC_REAL, ArgType1=IEC_UINT, Inline=Yes)
    INT_TO_REAL = ToFloat(:$[1]:) (ReturnType=IEC_REAL, ArgType1=IEC_INT, Inline=Yes)
    UDINT_TO_REAL = ToFloat(:$[1]:) (ReturnType=IEC_REAL, ArgType1=IEC_UDINT, Inline=Yes)
    DINT_TO_REAL = ToFloat(:$[1]:) (ReturnType=IEC_REAL, ArgType1=IEC_DINT, Inline=Yes)
    LREAL_TO_REAL = ToFloat(:$[1]:) (ReturnType=IEC_REAL, ArgType1=IEC_LREAL, Inline=Yes)
    TIME_TO_REAL = ToFloat(:$[1]:) (ReturnType=IEC_REAL, ArgType1=IEC_TIME, Inline=Yes)
    BOOL_TO_LREAL = ToLReal(:$[1]:) (ReturnType=IEC_LREAL, ArgType1=IEC_BOOL, Inline=Yes)
    USINT_TO_LREAL = ToLReal(:$[1]:) (ReturnType=IEC_LREAL, ArgType1=IEC_USINT, Inline=Yes)
    SINT_TO_LREAL = ToLReal(:$[1]:) (ReturnType=IEC_LREAL, ArgType1=IEC_SINT, Inline=Yes)
    UINT_TO_LREAL = ToLReal(:$[1]:) (ReturnType=IEC_LREAL, ArgType1=IEC_UINT, Inline=Yes)
    INT_TO_LREAL = ToLReal(:$[1]:) (ReturnType=IEC_LREAL, ArgType1=IEC_INT, Inline=Yes)
    UDINT_TO_LREAL = ToLReal(:$[1]:) (ReturnType=IEC_LREAL, ArgType1=IEC_UDINT, Inline=Yes)
    DINT_TO_LREAL = ToLReal(:$[1]:) (ReturnType=IEC_LREAL, ArgType1=IEC_DINT, Inline=Yes)
    REAL_TO_LREAL = ToLReal(:$[1]:) (ReturnType=IEC_LREAL, ArgType1=IEC_REAL, Inline=Yes)
    TIME_TO_LREAL = ToLReal(:$[1]:) (ReturnType=IEC_LREAL, ArgType1=IEC_TIME, Inline=Yes)
    BOOL_TO_STRING = ToString(:ToBool(:$[1]:):) (ReturnType=IEC_STRING, ArgType1=IEC_BOOL, Inline=Yes)
    USINT_TO_STRING = ToString(:ToUInt(:$[1],1:):) (ReturnType=IEC_STRING, ArgType1=IEC_USINT, Inline=Yes)
    SINT_TO_STRING = ToString(:ToInt(:$[1],1:):) (ReturnType=IEC_STRING, ArgType1=IEC_SINT, Inline=Yes)
    UINT_TO_STRING = ToString(:ToUInt(:$[1],2:):) (ReturnType=IEC_STRING, ArgType1=IEC_UINT, Inline=Yes)
    INT_TO_STRING = ToString(:ToInt(:$[1],2:):) (ReturnType=IEC_STRING, ArgType1=IEC_INT, Inline=Yes)
    UDINT_TO_STRING = ToString(:ToUInt(:$[1]:):) (ReturnType=IEC_STRING, ArgType1=IEC_UDINT, Inline=Yes)
    DINT_TO_STRING = ToString(:ToInt(:$[1]:):) (ReturnType=IEC_STRING, ArgType1=IEC_DINT, Inline=Yes)
    REAL_TO_STRING = ToString(:ToFloat(:$[1]:):) (ReturnType=IEC_STRING, ArgType1=IEC_REAL, Inline=Yes)
    LREAL_TO_STRING = ToString(:ToLReal(:$[1]:):) (ReturnType=IEC_STRING, ArgType1=IEC_LREAL, Inline=Yes)
    STRING_TO_BOOL = ToBool(:StrToInt(:$[1]:):) (ReturnType=IEC_BOOL, ArgType1=IEC_STRING, Inline=Yes)
    STRING_TO_USINT = ToUInt(:StrToInt(:$[1]:),1:) (ReturnType=IEC_USINT, ArgType1=IEC_STRING, Inline=Yes)
    STRING_TO_SINT = ToInt(:StrToInt(:$[1]:),1:) (ReturnType=IEC_SINT, ArgType1=IEC_STRING, Inline=Yes)
    STRING_TO_UINT = ToUInt(:StrToInt(:$[1]:),2:) (ReturnType=IEC_UINT, ArgType1=IEC_STRING, Inline=Yes)
    STRING_TO_INT = ToInt(:StrToInt(:$[1]:),2:) (ReturnType=IEC_INT, ArgType1=IEC_STRING, Inline=Yes)
    STRING_TO_UDINT = ToUInt(:StrToInt(:$[1]:):) (ReturnType=IEC_UDINT, ArgType1=IEC_STRING, Inline=Yes)
    STRING_TO_DINT = ToInt(:StrToInt(:$[1]:):) (ReturnType=IEC_DINT, ArgType1=IEC_STRING, Inline=Yes)
    STRING_TO_REAL = ToFloat(:ToLReal(:$[1]:):) (ReturnType=IEC_REAL, ArgType1=IEC_STRING, Inline=Yes)
    STRING_TO_LREAL = ToLReal(:$[1]:) (ReturnType=IEC_LREAL, ArgType1=IEC_STRING, Inline=Yes)
    LEN = __LEN(:$[1]:) (ReturnType=IEC_INT, ArgType1=IEC_STRING, Inline=Yes)
    LEFT = __LEFT(:$[1], $[2]:) (ReturnType=IEC_STRING, ArgType1=IEC_STRING, ArgType2=IEC_INT, Inline=Yes)
    RIGHT = __RIGHT(:$[1], $[2]:) (ReturnType=IEC_STRING, ArgType1=IEC_STRING, ArgType2=IEC_INT, Inline=Yes)
    MID = __MID(:$[1], $[2], $[3]:) (ReturnType=IEC_STRING, ArgType1=IEC_STRING, ArgType2=IEC_INT, ArgType3=IEC_INT, Inline=Yes)
    CONCAT = __CONCAT(:$[1], $[2]:) (ReturnType=IEC_STRING, ArgType1=IEC_STRING, ArgType2=IEC_STRING, Inline=Yes)
    INSERT = __INSERT(:$[1], $[2], $[3]:) (ReturnType=IEC_STRING, ArgType1=IEC_STRING, ArgType2=IEC_STRING, ArgType3=IEC_INT, Inline=Yes)
    DELETE = __DELETE(:$[1], $[2], $[3]:) (ReturnType=IEC_STRING, ArgType1=IEC_STRING, ArgType2=IEC_INT, ArgType3=IEC_INT, Inline=Yes)
    REPLACE = __REPLACE(:$[1], $[2], $[3], $[4]:) (ReturnType=IEC_STRING, ArgType1=IEC_STRING, ArgType2=IEC_STRING, ArgType3=IEC_INT, ArgType4=IEC_INT, Inline=Yes)
    FIND = __FIND(:$[1], $[2]:) (ReturnType=IEC_INT, ArgType1=IEC_STRING, ArgType2=IEC_STRING, Inline=Yes)
    IP_INST_NUM = IpInstNum(::) (ReturnType=IEC_INT, NumArgs=0)
    IP_OWNER_ID = IpOwnerId(::) (ReturnType=IEC_INT, NumArgs=0)
    PACKET_DATA_ADR = GetIpInt(:6:) (ReturnType=IEC_UDINT, NumArgs=0, Inline=Yes)
    PACKET_COMMAND_ADR = GetIpInt(:7:) (ReturnType=IEC_UDINT, NumArgs=0, Inline=Yes)
  Parameters:
    QUOTED (QuotedName=$R, ValueType=FLOAT, ReturnType=IEC_LREAL)
      ARG (ref=EXPR, DataType=INT, MinValue=0, MaxValue=999)
    QUOTED (QuotedName=$P, ValueType=FLOAT, ReturnType=IEC_LREAL)
      ARG (ref=EXPR, DataType=INT, MinValue=0, MaxValue=999)
    QUOTED (QuotedName=$EXB, ValueType=INT, ReturnType=IEC_SINT)
      ARG (ref=EXPR, DataType=INT, MinValue=0, MaxValue=99)
    QUOTED (QuotedName=$EXW, ValueType=INT, ReturnType=IEC_INT)
      ARG (ref=EXPR, DataType=INT, MinValue=0, MaxValue=99)
    QUOTED (QuotedName=$EXL, ValueType=INT, ReturnType=IEC_DINT)
      ARG (ref=EXPR, DataType=INT, MinValue=0, MaxValue=99)
    QUOTED (QuotedName=$EXF, ValueType=FLOAT, ReturnType=IEC_REAL)
      ARG (ref=EXPR, DataType=INT, MinValue=0, MaxValue=3999)
    QUOTED (QuotedName=$MW, Synchronous=Yes, ValueType=INT, ReturnType=IEC_INT)
      ARG (ref=EXPR, DataType=INT, MinValue=0, MaxValue=99)
    QUOTED (QuotedName=$ML, Synchronous=Yes, ValueType=INT, ReturnType=IEC_DINT)
      ARG (ref=EXPR, DataType=INT, MinValue=0, MaxValue=99)
    QUOTED (QuotedName=$MF, Synchronous=Yes, ValueType=FLOAT, ReturnType=IEC_REAL)
      ARG (ref=EXPR, DataType=INT, MinValue=0, MaxValue=99)
  ParserData (NestedComments=No, DefaultCaseSensitive=Yes, CommentsSpanLines=Yes, ReadWholeFileBeforeParsing=Yes, ExpectMainProgStmts=No, UseFubTemplates=No, LexerType=IEC, RuntimePreventOverflow=No, RoundRealToInt=No, AllowArrayRefWithoutIndex=Yes, DeclareEnumLiteralsAsConstants=No, AllowVariableAutoDereference=Yes, AllowStructMemberAutoDereference=No, AllowPassByRefFnArgAutoReference=No, AllowNamedFnArgs=Yes, AllowUnnamedFnArgs=Yes, AllowFnArgMixedNaming=Yes, AllowFnArgsOutOfSequence=No, AllowBuiltinFnArgsOutOfSequence=Yes, AllowFnArgsOmmitted=Yes, AllowIgnoredFnReturn=Yes, AllowIgnoredExtraSubArgs=No, AllowFnStringInputArgsShort=No, RefuseBuiltinFnUnknownArgName=Yes, AllowBuiltinFnArgCaseSensitive=Yes)
    TKG_OPEN_COMMENT = (*
    TKG_CLOSE_COMMENT = *)
    TKG_IEC_LINE_COMMENT = //
    TKG_TRUE = TRUE:[^\w\d] (IsPattern=Yes)
    TKG_FALSE = FALSE:[^\w\d] (IsPattern=Yes)
    TKG_PRIM_TYPE (IsPattern=Yes)
    TKG_OPEN_BRACKET = (
    TKG_CLOSE_BRACKET = )
    TKG_OPEN_INDEXBRACKET = [
    TKG_CLOSE_INDEXBRACKET = ]
    TKG_COMMA = ,
    TKG_SUBRANGE = ..
    TKG_IEC_BINARY_INTEGER = 2#_[01][01_]+|2#[01][01_]+|2#_[01]|2#[01] (IsPattern=Yes)
    TKG_IEC_OCTAL_INTEGER = 8#_[0-7][0-7_]+|8#[0-7][0-7_]+|8#_[0-7]|8#[0-7] (IsPattern=Yes)
    TKG_IEC_HEX_INTEGER = 16#_[\da-fA-F][\da-fA-F]+|16#[\da-fA-F][\da-fA-F_]+|16#_[\da-fA-F]|16#[\da-fA-F] (IsPattern=Yes)
    TKG_REAL = \d[\d_]*\.[\d_]+[Ee][\+\-]\d[\d_]*|\d[\d_]*\.[\d_]+[Ee]\d[\d_]*|\d[\d_]*\.[\d_]+ (IsPattern=Yes)
    TKG_REAL_EXP = \d[\d_]*[Ee]\d[\d_]*|\d[\d_]*[Ee][\+\-]\d[\d_]* (IsPattern=Yes)
    TKG_INTEGER = \d|\d[\d_]+ (IsPattern=Yes)
    TKG_DOT = .
    TKG_PATHSYNCH_REC_IEC = DO_PATH_SYNCH:[^\w\d] (IsPattern=Yes, EndRuleToken=Yes)
    TKG_PATHSYNCH_END = END_PATH_SYNCH:[^\w\d] (IsPattern=Yes, EndRuleToken=Yes)
    TKG_PATHSYNCH_IPEVAL = IP_EVAL:[^\w\d] (IsPattern=Yes)
    TKG_CYCLIC_PATHSYNCH_BLOCKING_IEC = CYCLIC_PS_BL:[^\w\d] (IsPattern=Yes, EndRuleToken=Yes)
    TKG_CYCLIC_PATHSYNCH_IEC = CYCLIC_PS:[^\w\d] (IsPattern=Yes, EndRuleToken=Yes)
    TKG_CYCLIC_BLOCKING_IEC = CYCLIC_BL:[^\w\d] (IsPattern=Yes, EndRuleToken=Yes)
    TKG_CYCLIC_IEC = CYCLIC:[^\w\d] (IsPattern=Yes, EndRuleToken=Yes)
    TKG_CYCLIC_END_IEC = END_CYCLIC:[^\w\d] (IsPattern=Yes, EndRuleToken=Yes)
    TKG_REFERENCE = REFERENCE:[^\w\d] (FollowedBy=TKG_IEC_TO, IsPattern=Yes)
    TKG_IEC_TO = TO:[^\w\d] (IsPattern=Yes)
    TKG_IEC_DO = DO:[^\w\d] (IsPattern=Yes, EndRuleToken=Yes)
    TKG_FOR_NOFINALDEC = FOR:[^\w\d] (FileXLInvalid=Yes, IsPattern=Yes)
    TKG_FORSTEP = BY:[^\w\d] (FileXLInvalid=Yes, IsPattern=Yes)
    TKG_ENDFOR = END_FOR:[^\w\d] (FileXLInvalid=Yes, IsPattern=Yes, EndRuleToken=Yes)
    TKG_IF = IF:[^\w\d] (IsPattern=Yes)
    TKG_THEN = THEN:[^\w\d] (IsPattern=Yes, EndRuleToken=Yes)
    TKG_BLOCK_ELSEIF = ELSIF:[^\w\d] (IsPattern=Yes)
    TKG_ELSE_AND_DEFAULT = ELSE:[^\w\d] (IsPattern=Yes, EndRuleToken=Yes)
    TKG_BLOCK_ENDIF = END_IF:[^\w\d] (IsPattern=Yes, EndRuleToken=Yes)
    TKG_SWITCH = CASE:[^\w\d] (IsPattern=Yes, FileXLInvalid=Yes)
    TKG_ENDSWITCH_NOBREAK = END_CASE:[^\w\d] (FileXLInvalid=Yes, IsPattern=Yes, EndRuleToken=Yes)
    TKG_WHILE = WHILE:[^\w\d] (FileXLInvalid=Yes, IsPattern=Yes)
    TKG_ENDWHILE = END_WHILE:[^\w\d] (FileXLInvalid=Yes, IsPattern=Yes, EndRuleToken=Yes)
    TKG_DO = REPEAT:[^\w\d] (FileXLInvalid=Yes, IsPattern=Yes, EndRuleToken=Yes)
    TKG_ENDDO_UNTIL = UNTIL:[^\w\d] (FileXLInvalid=Yes, IsPattern=Yes)
    TKG_ENDDO_POSTCOND = END_REPEAT:[^\w\d] (FileXLInvalid=Yes, IsPattern=Yes, EndRuleToken=Yes)
    TKG_BREAK = EXIT:[^\w\d] (FileXLInvalid=Yes, IsPattern=Yes)
    TKG_RETURN = RETURN:[^\w\d] (FileXLInvalid=Yes, IsPattern=Yes)
    TKG_IEC_SEL_FN = SEL:[^\w\d] (FileXLInvalid=Yes, IsPattern=Yes)
    TKG_IEC_MUX_FN = MUX:[^\w\d] (FileXLInvalid=Yes, IsPattern=Yes)
    TKG_TIME_LITERAL = time#\-[dDhHmMsS_\.\d]+|time#[dDhHmMsS_\.\d]+|t#\-[dDhHmMsS_\.\d]+|t#[dDhHmMsS_\.\d]+ (CaseSensitive=no, IsPattern=yes)
    TKG_DATE_AND_TIME_LITERAL = DT#[12]\d\d\d\-[\d\:\-]*|DATE_AND_TIME#[12]\d\d\d\-[\d\:\-]* (CaseSensitive=no, IsPattern=yes)
    TKG_DATE_LITERAL = D#[12]\d\d\d\-[\d\-]*|DATE#[12]\d\d\d\-[\d\-]* (CaseSensitive=no, IsPattern=yes)
    TKG_TIME_OF_DAY_LITERAL = TOD#\d[\d\:\.]*|TIME_OF_DAY#\d[\d\:\.]* (CaseSensitive=no, IsPattern=yes)
    TKG_ASSIGN_EQ = :=
    TKG_OPEN_IP_EXTENSION = {
    TKG_CLOSE_IP_EXTENSION = }
    TKG_IEC_OPEN_TYPE = TYPE:[^\w\d] (IsPattern=Yes)
    TKG_IEC_CLOSE_TYPE = END_TYPE:[^\w\d] (IsPattern=Yes, EndRuleToken=Yes)
    TKG_VAR = VAR:[^\w\d] (IsPattern=Yes)
    TKG_VAR_GLOBAL = VAR_GLOBAL:[^\w\d] (IsPattern=Yes)
    TKG_VAR_INPUT = VAR_INPUT:[^\w\d] (IsPattern=Yes)
    TKG_VAR_OUTPUT = VAR_OUTPUT:[^\w\d] (IsPattern=Yes)
    TKG_VAR_IN_OUT = VAR_IN_OUT:[^\w\d] (IsPattern=Yes)
    TKG_VAR_END = END_VAR:[^\w\d] (IsPattern=Yes, EndRuleToken=Yes)
    TKG_VAR_RETAIN = RETAIN:[^\d\w] (IsPattern=Yes)
    TKG_IP_RETAIN = IP_RETAIN:[^\d\w] (IsPattern=Yes)
    TKG_AT = AT:[^\d\w] (IsPattern=Yes)
    TKG_PLC = PLC:[^\d\w] (IsPattern=Yes)
    TKG_PV_UNDECL = UNRETAIN_VAR:[^\d\w] (IsPattern=Yes)
    TKG_VARSYNCH_IP = IP_SYNCH:[^\d\w] (IsPattern=Yes)
    TKG_VARSYNCH_PATH = PATH_SYNCH:[^\d\w] (IsPattern=Yes)
    TKG_CONSTANT = CONSTANT:[^\d\w] (IsPattern=Yes)
    TKG_VARSCOPE_IP_GLOBAL = IP_GLOBAL:[^\w\d] (IsPattern=Yes)
    TKG_VARSCOPE_SHARED_IP_GLOBAL = SHARED_IP_GLOBAL:[^\w\d] (IsPattern=Yes)
    TKG_VARSCOPE_NC_GLOBAL = NC_GLOBAL:[^\w\d] (IsPattern=Yes)
    TKG_VARSCOPE_PLC_GLOBAL = PLC_GLOBAL:[^\w\d] (IsPattern=Yes)
    TKG_VARSCOPE_IP_LOCAL = LOCAL:[^\w\d] (IsPattern=Yes)
    TKG_IEC_DATATYPE_SPEC = : (IsPattern=No)
    TKG_IEC_ARRAY = ARRAY:[^\w\d] (IsPattern=Yes)
    TKG_IEC_OF = OF:[^\w\d] (IsPattern=Yes)
    TKG_IEC_DELIM = ; (EndRuleToken=Yes)
    TKG_IEC_OPEN_STRUCT = STRUCT:[^\w\d] (IsPattern=Yes)
    TKG_IEC_CLOSE_STRUCT = END_STRUCT:[^\w\d] (IsPattern=Yes)
    TKG_BITWISE_LP_BINARY_AND = AND:[^\w\d] (IsPattern=Yes)
    TKG_BITWISE_LP_BINARY_OR = OR:[^\w\d] (IsPattern=Yes)
    TKG_BITWISE_LP_BINARY_XOR = XOR:[^\w\d] (IsPattern=Yes)
    TKG_BITWISE_UNARY_COMPLEMENT = NOT:[^\w\d] (IsPattern=Yes)
    TKG_COMP_EXACT_BINARY_GREATER_THAN_OR_EQ = >=
    TKG_COMP_EXACT_BINARY_LESS_THAN_OR_EQ = <=
    TKG_COMP_EXACT_BINARY_EQUAL_TO = =
    TKG_COMP_EXACT_BINARY_NOT_EQUAL_TO = <>
    TKG_COMP_EXACT_BINARY_GREATER_THAN = >
    TKG_COMP_EXACT_BINARY_LESS_THAN = <
    TKG_ARITH_BINARY_PLUS = +
    TKG_ARITH_BINARY_MINUS = -
    TKG_ARITH_BINARY_POWER = **
    TKG_ARITH_BINARY_MULTIPLY = *
    TKG_ARITH_BINARY_DIVIDE = /
    TKG_ARITH_BINARY_MODULO = MOD:[^\w\d] (IsPattern=Yes)
    TKG_PRAGMA = #pragma:[^\w\d] (IsPattern=Yes, FollowedBy=TKG_IDENTIFIER)
    TKG_INCLUDE = #include:[^\w\d] (IsPattern=Yes)
    TKG_PROG_START = PROGRAM:[^\w\d] (IsPattern=Yes, FollowedBy=TKG_PROG_NAME)
    TKG_PROG_NAME = _INIT:[^\w\d]|_CYCLIC:[^\w\d]|_EXIT:[^\w\d]|_MAIN:[^\w\d] (IsPattern=Yes, EndRuleToken=Yes)
    TKG_PROG_END = END_PROGRAM:[^\w\d] (IsPattern=Yes, EndRuleToken=Yes)
    TKG_SUBPROG_START = FUNCTION:[^\w\d] (IsPattern=Yes)
    TKG_SUBPROG_END = END_FUNCTION:[^\w\d] (IsPattern=Yes, EndRuleToken=Yes)
    TKG_FUB_DECL = FUNCTION_BLOCK:[^\w\d] (IsPattern=Yes)
    TKG_FUB_END = END_FUNCTION_BLOCK:[^\w\d] (IsPattern=Yes, EndRuleToken=Yes)
    TKG_RETURN = RETURN:[^\w\d] (IsPattern=Yes)
    TKG_ACCESS = ACCESS:[^\w\d] (IsPattern=Yes)
    TKG_DEREF_OP = ^
    TKG_ACTION = ACTION:[^\w\d] (IsPattern=Yes)
    TKG_ACTION_END = END_ACTION:[^\w\d] (IsPattern=Yes, EndRuleToken=Yes)
    TKG_IEC_TYPED_VALUE = \w#:[\w\d\+\-]|\w[\w\d]+#:[\w\d\+\-] (IsPattern=Yes)
    TKG_PARAM_PREFIX = $R:[^\w\d]|$P:[^\w\d]|$MW:[^\w\d]|$ML:[^\w\d]|$MF:[^\w\d]|$EXW:[^\w\d]|$EXL:[^\w\d]|$EXF:[^\w\d]|$EXB:[^\w\d] (IsPattern=Yes)
    TKG_IDENTIFIER = \w|\w[\w\d$]+|$[\w\d$]+ (IsPattern=Yes)
    TKG_INIT_IDENTIFIER = \w|\w[\w\d$]+|$[\w\d$]+ (IsPattern=Yes, Disabled=Yes)
  StringChars (AsciiStringStart=', AsciiStringEnd=', UTF16StringStart=", UTF16StringEnd=")
    EscapeSeq (Search=$N, CaseSensitive=Yes, ReplaceValue=10)
    EscapeSeq (Search=$n, CaseSensitive=Yes, ReplaceValue=10)
    EscapeSeq (Search=$L, CaseSensitive=Yes, ReplaceValue=10)
    EscapeSeq (Search=$l, CaseSensitive=Yes, ReplaceValue=10)
    EscapeSeq (Search=$P, CaseSensitive=Yes, ReplaceValue=12)
    EscapeSeq (Search=$p, CaseSensitive=Yes, ReplaceValue=12)
    EscapeSeq (Search=$R, CaseSensitive=Yes, ReplaceValue=13)
    EscapeSeq (Search=$r, CaseSensitive=Yes, ReplaceValue=13)
    EscapeSeq (Search=$T, CaseSensitive=Yes, ReplaceValue=9)
    EscapeSeq (Search=$t, CaseSensitive=Yes, ReplaceValue=9)
    EscapeSeq (Search=$', CaseSensitive=Yes, ReplaceStr=')
    EscapeSeq (Search=$", CaseSensitive=Yes, ReplaceStr=")
    EscapeSeq (Search=$[\dA-Fa-f]+, IsPattern=Yes, CaseSensitive=Yes, ReplaceEncodingBase=16)
    EscapeSeq (Search=$$, ReplaceStr=$)
    EscapeSeq (Search=$, ReplaceStr=)
```

### Data object Logical/MotionHandling/Interpreter/GmcIpConfig/gmciplog (Cnc, version 2.47.4)
